// POUs/IO/Drives/SoE/Ax5000ParamSTRUCTs/P/AX5000_P_0270
{attribute 'pack_mode' := '1'}//Ensures 1-byte-alignmend
TYPE AX5000_P_0270 :
STRUCT
	Actual_lenght:UINT;
	Max_lenght:UINT;
	Feedback1:STRING(29);
//	{attribute 'hide'}
	Rsvd1:UINT;
	Serial_number_feedback1:ARRAY[0..1] OF UDINT;
	Feedback2:STRING(29);
//	{attribute 'hide'}
	Rsvd2:UINT;
	Serial_number_feedback2:ARRAY[0..1] OF UDINT;
	Modulo_value:UDINT;

(*Data read from file*)

(*data[0][0]*)
	Feedback_number1:UINT;
	Data_set1:UINT;
	Feedback_position1:UDINT;
	Modulo_position1:UDINT;
	Crc1:UDINT;
(*data[0][1]*)
	Feedback_number2:UINT;
	Data_se2t:UINT;
	Feedback_position2:UDINT;
	Modulo_position2:UDINT;
	Crc2:UDINT;
(*data[1][0]*)
	Feedback_number3:UINT;
	Data_set3:UINT;
	Feedback_position3:UDINT;
	Modulo_position3:UDINT;
	Crc3:UDINT;
(*data[1][1]*)
	Feedback_number4:UINT;
	Data_set4:UINT;
	Feedback_position4:UDINT;
	Modulo_position4:UDINT;
	Crc4:UDINT;


(*Current Data*)


(*data[0][0]*)
	Feedback_number5:UINT;
	Data_set5:UINT;
	Feedback_position5:UDINT;
	Modulo_position5:UDINT;
	Crc5:UDINT;
(*data[0][1]*)
	Feedback_number6:UINT;
	Data_se6t:UINT;
	Feedback_position6:UDINT;
	Modulo_position:UDINT;
	Crc6:UDINT;
(*data[1][0]*)
	Feedback_number7:UINT;
	Data_set7:UINT;
	Feedback_position7:UDINT;
	Modulo_position7:UDINT;
	Crc7:UDINT;
(*data[1][1]*)
	Feedback_number8:UINT;
	Data_set8:UINT;
	Feedback_position8:UDINT;
	Modulo_position8:UDINT;
	Crc8:UDINT;
END_STRUCT
END_TYPE

// POUs/IO/Drives/SoE/Ax5000ParamSTRUCTs/P/AX5000_P_0271
TYPE AX5000_P_0271 :
STRUCT
	Save_sosition_offset_pc:UINT;
END_STRUCT
END_TYPE

// POUs/IO/Drives/SoE/Ax5000ParamSTRUCTs/P/AX5000_P_0272
{attribute 'pack_mode' := '1'}//Ensures 1-byte-alignmend
TYPE AX5000_P_0272 :
STRUCT
	Actual_Length : UINT := 8;
	Max_Length : UINT := 8;
	(* FeedbackNumber &amp; MemorySelection *)
	Data : BYTE;
//	{attribute 'hide'}
	Rsvd1 : ARRAY [1..3] OF USINT;
	Position_Offset : UDINT;	
END_STRUCT
END_TYPE

// POUs/IO/Drives/SoE/Ax5000ParamSTRUCTs/P/AX5000_P_0273
TYPE AX5000_P_0273 EXTENDS ST_AX5000_P_0273:
STRUCT
(*
	Actual_lenght:UINT:= 112;
	Max_lenght:UINT := 112;
(*feedback 1*)
 {attribute 'GUID' := 'D1EB669D-3061-44CC-A2EE-FBF75E3AC2F6'}
 {attribute 'Namespace' := 'AX5000'}
Feedback1 : ST_AX5000_P_0273_Feedback;
(*
(*Encoder Memory*)
	Data_valid1:UINT;
//	{attribute 'hide'}
	rsvd1:UINT;
	Position_offset1:UDINT;
(*Drive Memory*)
	Data_valid2:UINT;
//	{attribute 'hide'}
	rsvd2:UINT;
	Feedback_type1:STRING(29);
//	{attribute 'hide'}
	rsvd3:UINT;
	Feedback_serial_number:ARRAY[0..1]OF UDINT;
	Position_offset2:UDINT;
*)
(*feedback 2*)
{attribute 'GUID' := 'D1EB669D-3061-44CC-A2EE-FBF75E3AC2F6'}
 {attribute 'Namespace' := 'AX5000'}
Feedback2 : ST_AX5000_P_0273_Feedback;
(*
(*Encoder Memory*)
	Data_valid3:UINT;
//	{attribute 'hide'}
	rsvd4:UINT;
	Position_offset3:UDINT;
(*Drive Memory*)
	Data_valid4:UINT;
//	{attribute 'hide'}
	rsvd5:UINT;
	Feedback_type2:STRING(29);
//	{attribute 'hide'}
	rsvd6:UINT;
	Feedback_serial_number2:ARRAY[0..1]OF UDINT;
	Position_offset4:UDINT;
*)	

//	{attribute 'hide'}
	Rsvd1 : UDINT;
*)
END_STRUCT
END_TYPE

// POUs/IO/Drives/SoE/Ax5000ParamSTRUCTs/P/AX5000_P_0274
{attribute 'pack_mode' := '1'}
TYPE AX5000_P_0274 :
STRUCT
	Actual_lenght:UINT;
	Max_lenght:UINT;
	Position_offset_feedback_1:UDINT;
	Position_offset_feedback_2:UDINT;
END_STRUCT
END_TYPE

// POUs/IO/Drives/SoE/Ax5000ParamSTRUCTs/P/AX5000_P_0275
TYPE AX5000_P_0275 EXTENDS ST_AX5000_P_0275: 
	STRUCT
(*		 {attribute 'GUID' := 'A39361D3-D4AC-4F67-8FEE-F366F3137B89'}
		 {attribute 'Namespace' := 'AX5000'}
		ActiveFeedbackAndMemory : E_AX5000_P_0275_ActiveFeedbackAndMemory;
		InitializationErrorBehavior : BIT;
		 {attribute 'hide'}
		_reserved1 : BIT;
		 {attribute 'hide'}
		_reserved2 : BIT;
		 {attribute 'hide'}
		_reserved3 : BIT;
		 {attribute 'hide'}
		_reserved4 : BIT;
		 {attribute 'hide'}
		_reserved5 : BIT;
		 {attribute 'hide'}
		_reserved6 : BIT;
		 {attribute 'hide'}
		_reserved7 : BIT;
*)
	END_STRUCT
END_TYPE

// POUs/IO/Drives/SoE/Ax5000ParamSTRUCTs/P/AX5000_P_0276
TYPE AX5000_P_0276 :
STRUCT
	Data_storage_feedback1_Data_storge_feedback2:UDINT;	(*Data_storage_feedback1 8Bit; Data_storage_feedback2 8 Bit*)
END_STRUCT
END_TYPE

// POUs/IO/Drives/SoE/Ax5000ParamSTRUCTs/P/AX5000_P_0277
TYPE AX5000_P_0277 :
STRUCT
	Schedule_modulo_init_data_saving:UINT;
END_STRUCT
END_TYPE

// POUs/IO/Drives/SoE/Ax5000ParamSTRUCTs/P/AX5000_P_0278
TYPE AX5000_P_0278 :
STRUCT
	Ignore_for_one_PreOp_SafeOp_transition:UINT;
END_STRUCT
END_TYPE

// POUs/IO/Drives/SoE/Ax5000ParamSTRUCTs/P/AX5000_P_0300
TYPE AX5000_P_0300 :
STRUCT
	Actual_lenght:UINT;
	Max_lenght:UINT;
	Error_number_history:ARRAY[0..99] OF UDINT;
END_STRUCT
END_TYPE

// POUs/IO/Drives/SoE/Ax5000ParamSTRUCTs/P/AX5000_P_0301
TYPE AX5000_P_0301 :
STRUCT
	Actual_lenght:UINT;
	Max_lenght:UINT;
	Error_times_history:ARRAY[0..99] OF UDINT;
END_STRUCT
END_TYPE

// POUs/IO/Drives/SoE/Ax5000ParamSTRUCTs/P/AX5000_P_0302
TYPE AX5000_P_0302 :
STRUCT
	Display_value_line_1:UINT;
END_STRUCT
END_TYPE

// POUs/IO/Drives/SoE/Ax5000ParamSTRUCTs/P/AX5000_P_0303
TYPE AX5000_P_0303 :
STRUCT
	Display_value_line_2:UINT;
END_STRUCT
END_TYPE

// POUs/IO/Drives/SoE/Ax5000ParamSTRUCTs/P/AX5000_P_0304
TYPE AX5000_P_0304 :
STRUCT
	Log_errors_Log_warnings_Log_information_rsvd:UINT;	(*Log_errors 1; BitLog_warnings 1; BitLog_information 1 Bit*)
END_STRUCT
END_TYPE

// POUs/IO/Drives/SoE/Ax5000ParamSTRUCTs/P/AX5000_P_0305
TYPE AX5000_P_0305 :
STRUCT
	I2C_Bus_Lcd_Ext_ADC_Encoder_parameter_channel_String_KeyPad_Procedure_command_calls_Powermanagement_Feedback_Dsp_Device_state_machine_rsvd:UDINT;
(*I2C_Bus 2 Bit; Lcd 2 Bit; Ext_ADC 2 Bit; Encoder 2 Bit; parameter_channel_String 2 Bit; KeyPad 2 Bit; Procedure_command_calls 2 Bit; Powermanagement 2 Bit; Feedback_Dsp 2 Bit; Device_state_machine 2 Bit; rsvd 12 Bit*)
END_STRUCT
END_TYPE

// POUs/IO/Drives/SoE/Ax5000ParamSTRUCTs/P/AX5000_P_0306
TYPE AX5000_P_0306 :
STRUCT
	Actual_main_loop_time:UINT;
END_STRUCT
END_TYPE

// POUs/IO/Drives/SoE/Ax5000ParamSTRUCTs/P/AX5000_P_0307
TYPE AX5000_P_0307 :
STRUCT
	Max_main_loop_time:UINT;
END_STRUCT
END_TYPE

// POUs/IO/Drives/SoE/Ax5000ParamSTRUCTs/P/AX5000_P_0308
TYPE AX5000_P_0308 :
STRUCT
	Actual_ctrl_loop_time:UINT;
END_STRUCT
END_TYPE

// POUs/IO/Drives/SoE/Ax5000ParamSTRUCTs/P/AX5000_P_0309
TYPE AX5000_P_0309 :
STRUCT
	Max_ctrl_loop_time:UINT;
END_STRUCT
END_TYPE

// POUs/IO/Drives/SoE/Ax5000ParamSTRUCTs/P/AX5000_P_0310
TYPE AX5000_P_0310 :
STRUCT
	Torque_off_Slow_down_according_Open_loop_ramp_Closed_loop_ramp_NC_handling_rsvd:UINT;
	(*Torque_off 1 Bit; Slow_down_according 1 Bit; Open_loop_ramp 1 Bit; Closed_loop_ramp 1 Bit; NC_handling  1 Bit;  rsvd  11 Bit; *)
END_STRUCT
END_TYPE

// POUs/IO/Drives/SoE/Ax5000ParamSTRUCTs/P/AX5000_P_0311
TYPE AX5000_P_0311 :
STRUCT
	PLL_ctrl_error:DINT;
END_STRUCT
END_TYPE

// POUs/IO/Drives/SoE/Ax5000ParamSTRUCTs/P/AX5000_P_0312
TYPE AX5000_P_0312 :
STRUCT
	PCB_temperature:UINT;
END_STRUCT
END_TYPE

// POUs/IO/Drives/SoE/Ax5000ParamSTRUCTs/P/AX5000_P_0313
TYPE AX5000_P_0313 :
STRUCT
	Actual_lenght:UINT;
	Max_lenght:UINT;
	String_output_mode:UINT;
	Backlight_mode:UINT;
	Keypad_mode:UINT;
//	{attribute 'hide'}
	Rsvd:UINT;
	Output_string:STRING(39);
END_STRUCT
END_TYPE

// POUs/IO/Drives/SoE/Ax5000ParamSTRUCTs/P/AX5000_P_0314
TYPE AX5000_P_0314 :
STRUCT
	Actual_lenght:UINT;
	Max_lenght:UINT;
	String_output_mode:UINT;
	Backlight_mode:UINT;
	Keypad_mode:UINT;
//	{attribute 'hide'}
	Rsvd:UINT;
	Output_string:STRING(39);
END_STRUCT
END_TYPE

// POUs/IO/Drives/SoE/Ax5000ParamSTRUCTs/P/AX5000_P_0315
TYPE AX5000_P_0315 :
STRUCT
	Configuration_Output_number_Set_output_error_Set_output_warning_rsvd:UINT;
	(*Configuration 3 Bit; Output_number 5 Bit; Set_output_error 1 Bit; Set_output_warning 1 Bit; rsvd 6 Bit; *)
END_STRUCT
END_TYPE

// POUs/IO/Drives/SoE/Ax5000ParamSTRUCTs/P/AX5000_P_0316
TYPE AX5000_P_0316 :
STRUCT
	Actual_lenght:UINT;
	Max_lenght:UINT;
	Mode:UINT;
	Level:UINT;		(*Decimal Point 1*)
END_STRUCT
END_TYPE

// POUs/IO/Drives/SoE/Ax5000ParamSTRUCTs/P/AX5000_P_0317
TYPE AX5000_P_0317 :
STRUCT
	Actual_amplifier_stilisation:UDINT;
END_STRUCT
END_TYPE

// POUs/IO/Drives/SoE/Ax5000ParamSTRUCTs/P/AX5000_P_0320
TYPE AX5000_P_0320 EXTENDS ST_AX5000_P_0320:
STRUCT
(*	Actual_lenght:UINT;
	Max_lenght:UINT;
	Firmware_version:UINT;
	Firmware_build:UINT;
	Bootloader_build:UINT;
	MainDsp_compiler_version:UDINT;
	FeedbackDsp_compiler_version:UDINT;
	Option_card_firmware_version:UINT;
	Option_card_firmware_build:UINT;
	Option_card_interface:UINT;
//	{attribute 'hide'}
	Rsvd:UDINT;
	Option_card_Dsp_compiler_version:UDINT;
	Intf_Build_Version:UINT;
//	{attribute 'hide'}
	Rsvd2:UINT;
//	{attribute 'hide'}
	Rsvd3:UINT;
*)
END_STRUCT
END_TYPE

// POUs/IO/Drives/SoE/Ax5000ParamSTRUCTs/P/AX5000_P_0321
{attribute 'pack_mode' := '1'}
TYPE AX5000_P_0321 :
STRUCT
	Actual_lenght:UINT;
	Max_lenght:UINT;
	Disc_size:UDINT;
	Usend_size:UDINT;
	Alignment:UDINT;
	Free_size:UDINT;
(*File 0*)
	Type0:UINT;
//	{attribute 'hide'}
	rsvd0:UINT;
	Version0:UINT;
	Build0:UINT;
	Time_H0:UDINT;
	Time_L0:UDINT;
	Id10:UINT;
	Id20:UINT;
	Size0:UDINT;
	Size_on_disk0:UDINT;
	alignment0:UDINT;
	Start_adresse0:UDINT;

(*File 1*)
	Type1:UINT;
//	{attribute 'hide'}
	Rsvd1:UINT;
	Version1:UINT;
	Build1:UINT;
	Time_H1:UDINT;
	Time_L1:UDINT;
	Id11:UINT;
	Id21:UINT;
	Size1:UDINT;
	Size_on_disk1:UDINT;
	alignment1:UDINT;
	Start_adresse1:UDINT;

(*File 2*)
	Type2:UINT;
//	{attribute 'hide'}
	Rsvd2:UINT;
	Version2:UINT;
	Build2:UINT;
	Time_H2:UDINT;
	Time_L2:UDINT;
	Id12:UINT;
	Id22:UINT;
	Size2:UDINT;
	Size_on_disk2:UDINT;
	alignment2:UDINT;
	Start_adresse2:UDINT;

(*File 3*)
	Type3:UINT;
//	{attribute 'hide'}
	Rsvd3:UINT;
	Version3:UINT;
	Build3:UINT;
	Time_H3:UDINT;
	Time_L3:UDINT;
	Id13:UINT;
	Id23:UINT;
	Size3:UDINT;
	Size_on_disk3:UDINT;
	alignment3:UDINT;
	Start_adresse3:UDINT;

(*File 4*)
	Type4:UINT;
//	{attribute 'hide'}
	Rsvd4:UINT;
	Version4:UINT;
	Build4:UINT;
	Time_H4:UDINT;
	Time_L4:UDINT;
	Id14:UINT;
	Id24:UINT;
	Size4:UDINT;
	Size_on_disk4:UDINT;
	alignment4:UDINT;
	Start_adresse4:UDINT;

(*File 5*)
	Type5:UINT;
//	{attribute 'hide'}
	Rsvd5:UINT;
	Version5:UINT;
	Build5:UINT;
	Time_H5:UDINT;
	Time_L5:UDINT;
	Id15:UINT;
	Id25:UINT;
	Size5:UDINT;
	Size_on_disk5:UDINT;
	alignment5:UDINT;
	Start_adresse5:UDINT;

(*File 6*)
	Type6:UINT;
//	{attribute 'hide'}
	Rsvd6:UINT;
	Version6:UINT;
	Build6:UINT;
	Time_H6:UDINT;
	Time_L6:UDINT;
	Id16:UINT;
	Id26:UINT;
	Size6:UDINT;
	Size_on_disk6:UDINT;
	alignment6:UDINT;
	Start_adresse6:UDINT;

(*File 7*)
	Type7:UINT;
//	{attribute 'hide'}
	Rsvd7:UINT;
	Version7:UINT;
	Build7:UINT;
	Time_H7:UDINT;
	Time_L7:UDINT;
	Id17:UINT;
	Id27:UINT;
	Size7:UDINT;
	Size_on_disk7:UDINT;
	Alignment7:UDINT;
	Start_adresse7:UDINT;

(*File 8*)
	Type8:UINT;
//	{attribute 'hide'}
	Rsvd8:UINT;
	Version8:UINT;
	Build8:UINT;
	Time_H8:UDINT;
	Time_L8:UDINT;
	Id18:UINT;
	Id28:UINT;
	Size8:UDINT;
	Size_on_disk8:UDINT;
	Alignment8:UDINT;
	Start_adresse8:UDINT;

(*File 9*)
	Type9:UINT;
	Rsvd9:UINT;
	Version9:UINT;
	Build9:UINT;
	Time_H9:UDINT;
	Time_L9:UDINT;
	Id19:UINT;
	Id29:UINT;
	Size9:UDINT;
	Size_on_disk9:UDINT;
	alignment9:UDINT;
	Start_adresse9:UDINT;
END_STRUCT
END_TYPE

// POUs/IO/Drives/SoE/Ax5000ParamSTRUCTs/P/AX5000_P_0322
//	{attribute 'hide'}
TYPE AX5000_P_0322 :
STRUCT
	Actual_lenght:UINT;
	Max_lenght:UINT;


	PCB_ID_version:UINT;
	Hwld1:UINT;
	Hwld2:UINT;
	Hwld3:UINT;
	Manufacturing_Data:UINT;
	Serial_number_low:UINT;
	Serial_number_high:UINT;
	Checksum:UINT;


	PCB_ID_version1:UINT;
	Hwld4:UINT;
	Hwld5:UINT;
	Hwld6:UINT;
	Manufacturing_Data1:UINT;
	Serial_number_low1:UINT;
	Serial_number_high1:UINT;
	Checksum1:UINT;


	PCB_ID_version2:UINT;
	Hwld7:UINT;
	Hwld8:UINT;
	Hwld9:UINT;
	Manufacturing_Data2:UINT;
	Serial_number_low2:UINT;
	Serial_number_high2:UINT;
	Checksum2:UINT;


	PCB_ID_version3:UINT;
	Hwld10:UINT;
	Hwld11:UINT;
	Hwld12:UINT;
	Manufacturing_Data3:UINT;
	Serial_number_low3:UINT;
	Serial_number_high3:UINT;
	Checksum3:UINT;


	PCB_ID_version4:UINT;
	Hwld13:UINT;
	Hwld14:UINT;
	Hwld15:UINT;
	Manufacturing_Data4:UINT;
	Serial_number_low4:UINT;
	Serial_number_high4:UINT;
	Checksum4:UINT;


	PCB_ID_version5:UINT;
	Hwld16:UINT;
	Hwld17:UINT;
	Hwld18:UINT;
	Manufacturing_Data5:UINT;
	Serial_number_low5:UINT;
	Serial_number_high5:UINT;
	Checksum5:UINT;


	Control_Pcb_Id_valid:UINT;
	Power_Pcb_Id_valid:UINT;
	Driver_Pcb_Id_valid:UINT;
	Front_Pcb_Id_valid:UINT;
	OptionSlot_Pcb_Id_valid:UINT;
	SafetySlot_Id_valid:UINT;
	Dsp_Revidion:UINT;
	Dsp_Id_Xint_Revision:UINT;
	Feedback_Dsp_Id:UINT;
	Feedback_Dsp_Revision:UINT;
	Esc_Revision:UINT;
	Esc_build:UINT;
	Esc_type:UINT;
	FPGA_device_Type:UINT;
	FPGA_device_Subtype:UINT;
	FPGA_version_number:UINT;
	FPGA_build_number:UINT;
	Option_slot_FPGA:UINT;
END_STRUCT
END_TYPE

// POUs/IO/Drives/SoE/Ax5000ParamSTRUCTs/P/AX5000_P_0323
TYPE AX5000_P_0323 :
STRUCT
	Actual_lenght:UINT;
	Max_lenght:UINT;

(*control*)
	Total:UDINT;
	Available:UDINT;
	Total1:UDINT;
	Available1:UDINT;
	Total2:UDINT;
	Available2:UDINT;
	Total3:UDINT;
	Available3:UDINT;

(*front*)
	Total4:UDINT;
	Available4:UDINT;
	Total5:UDINT;
	Available5:UDINT;
	Total6:UDINT;
	Available6:UDINT;
	Total7:UDINT;
	Available7:UDINT;


(*option*)
	Toal8:UDINT;
	Available8:UDINT;
	Total9:UDINT;
	Available9:UDINT;
	Total10:UDINT;
	Available10:UDINT;
	Total11:UDINT;
	Available11:UDINT;
END_STRUCT
END_TYPE

// POUs/IO/Drives/SoE/Ax5000ParamSTRUCTs/P/AX5000_P_0324
TYPE AX5000_P_0324 :
STRUCT
	Actual_lenght:UINT;
	Max_lenght:UINT;
	ProductCode_RevisionNo:STRING;
END_STRUCT
END_TYPE

// POUs/IO/Drives/SoE/Ax5000ParamSTRUCTs/P/AX5000_P_0325
TYPE AX5000_P_0325 :
STRUCT
	Actual_lenght:UINT;
	Max_lenght:UINT;
	Compile_time_and_date:STRING;
END_STRUCT
END_TYPE

// POUs/IO/Drives/SoE/Ax5000ParamSTRUCTs/P/AX5000_P_0326
TYPE AX5000_P_0326 :
STRUCT
	Actual_lenght:UINT;
	Max_lenght:UINT;
	Release_note:STRING;
END_STRUCT
END_TYPE

// POUs/IO/Drives/SoE/Ax5000ParamSTRUCTs/P/AX5000_P_0350
TYPE AX5000_P_0350 EXTENDS ST_AX5000_P_0350: 
STRUCT
//	Error_reaction_Controlword:UINT;
END_STRUCT
END_TYPE

// POUs/IO/Drives/SoE/Ax5000ParamSTRUCTs/P/AX5000_P_0351
TYPE AX5000_P_0351 :
STRUCT
	Error_reaktion_delay_time:UINT;
END_STRUCT
END_TYPE

// POUs/IO/Drives/SoE/Ax5000ParamSTRUCTs/P/AX5000_P_0352
TYPE AX5000_P_0352 :
STRUCT
	Drive_halt_jerk_bipolar:UDINT;
END_STRUCT
END_TYPE

// POUs/IO/Drives/SoE/Ax5000ParamSTRUCTs/P/AX5000_P_0353
TYPE AX5000_P_0353 :
STRUCT
	Emergency_stop_jerk:UDINT;
END_STRUCT
END_TYPE

// POUs/IO/Drives/SoE/Ax5000ParamSTRUCTs/P/AX5000_P_0354
TYPE AX5000_P_0354 :
STRUCT
	Standstill_window_monitoring_time:UINT;
END_STRUCT
END_TYPE

// POUs/IO/Drives/SoE/Ax5000ParamSTRUCTs/P/AX5000_P_0356
//	{attribute 'hide'}
TYPE AX5000_P_0356 :
STRUCT
	Actual_lenght:UINT;
	Max_lenght:UINT;
//	{attribute 'hide'}
	Rsvd:UDINT;
	Available_for:UINT;
	Command_mode:UINT;
	Current_level:UINT;
	Current_slope:UINT;
	Wait_time_before_braking:UINT;
	First_phase_activation_time_with_f_f1:UINT;
	Rotary_field_frequency_f1:UINT;
	Rotor_slowdown_mode:UINT;
	Second_phase_activation_time_with_f_0Hz:UINT;
	Wait_ime_after_braking:UINT;
//	{attribute 'hide'}
	Rsvd1:UINT;
//	{attribute 'hide'}
	Rsvd2:UINT;
	Synchronus_motor:ARRAY[0..11] OF UINT;
END_STRUCT
END_TYPE

// POUs/IO/Drives/SoE/Ax5000ParamSTRUCTs/P/AX5000_P_0360
TYPE AX5000_P_0360 :
STRUCT
	Parameter_set_prearrangement:UINT;
END_STRUCT
END_TYPE

// POUs/IO/Drives/SoE/Ax5000ParamSTRUCTs/P/AX5000_P_0361
TYPE AX5000_P_0361 :
STRUCT
	Actual_lenght:UINT;
	Max_lenght:UINT;
	Parameter_set_configuration:ARRAY[0..34] OF UINT;
END_STRUCT
END_TYPE

// POUs/IO/Drives/SoE/Ax5000ParamSTRUCTs/P/AX5000_P_0400
TYPE AX5000_P_0400 EXTENDS ST_AX5000_P_0400:
STRUCT
//	Hardware_enable_configuration:UINT;
END_STRUCT
END_TYPE

// POUs/IO/Drives/SoE/Ax5000ParamSTRUCTs/P/AX5000_P_0401
TYPE AX5000_P_0401 :
STRUCT
	Positiv_limit_switch: ST_AX5000_P_0401_LimitSwitch;
	Negativ_limit_switch: ST_AX5000_P_0401_LimitSwitch;
END_STRUCT
END_TYPE

// POUs/IO/Drives/SoE/Ax5000ParamSTRUCTs/P/AX5000_P_0402
TYPE AX5000_P_0402 :
STRUCT
	Redy_to_operate_configuration:UINT;
END_STRUCT
END_TYPE

// POUs/IO/Drives/SoE/Ax5000ParamSTRUCTs/P/AX5000_P_0451
TYPE AX5000_P_0451 :
STRUCT
	Current_controller_settings:UINT;
END_STRUCT
END_TYPE

// POUs/IO/Drives/SoE/Ax5000ParamSTRUCTs/P/AX5000_P_0452
TYPE AX5000_P_0452 :
STRUCT
	Current_controller_control_word:UINT;
END_STRUCT
END_TYPE

// POUs/IO/Drives/SoE/Ax5000ParamSTRUCTs/P/AX5000_P_0453
TYPE AX5000_P_0453 :
STRUCT
	Current_controller_status_word:UINT;
END_STRUCT
END_TYPE

// POUs/IO/Drives/SoE/Ax5000ParamSTRUCTs/P/AX5000_P_0454
TYPE AX5000_P_0454 :
STRUCT
	Effective_torque_command_value:UINT;
END_STRUCT
END_TYPE

// POUs/IO/Drives/SoE/Ax5000ParamSTRUCTs/P/AX5000_P_0455
{attribute 'pack_mode' := '1'}
TYPE AX5000_P_0455 :
STRUCT
	Actual_lenght:UINT;
	Max_lenght:UINT;
	Mode:UINT;
	Rsvd:UINT;
	Min_voltage:UINT;
	Max_voltage:UINT;
	Max_current_for_fielweakening:UDINT;
	Max_velocity_for_fielweakening:UDINT;
END_STRUCT
END_TYPE

// POUs/IO/Drives/SoE/Ax5000ParamSTRUCTs/P/AX5000_P_0456
TYPE AX5000_P_0456 :
STRUCT
	Actual_motor_voltage_phase_U:UINT;
END_STRUCT
END_TYPE

// POUs/IO/Drives/SoE/Ax5000ParamSTRUCTs/P/AX5000_P_0457
TYPE AX5000_P_0457 :
STRUCT
	Actual_motor_voltage_phase_V:UINT;
END_STRUCT
END_TYPE

// POUs/IO/Drives/SoE/Ax5000ParamSTRUCTs/P/AX5000_P_0458
TYPE AX5000_P_0458 :
STRUCT
	Actual_motor_voltage_phase_W:UINT;
END_STRUCT
END_TYPE

// POUs/IO/Drives/SoE/Ax5000ParamSTRUCTs/P/AX5000_P_0459
TYPE AX5000_P_0459 :
STRUCT
	Actual_torquw_generating_current:UINT;
END_STRUCT
END_TYPE

// POUs/IO/Drives/SoE/Ax5000ParamSTRUCTs/P/AX5000_P_0460
TYPE AX5000_P_0460 :
STRUCT
	Actual_flux_generating_current:UINT;
END_STRUCT
END_TYPE

// POUs/IO/Drives/SoE/Ax5000ParamSTRUCTs/P/AX5000_P_0461
TYPE AX5000_P_0461 :
STRUCT
	Actual_absolute_current:UINT;
END_STRUCT
END_TYPE

// POUs/IO/Drives/SoE/Ax5000ParamSTRUCTs/P/AX5000_P_0462
TYPE AX5000_P_0462 :
STRUCT
	Actual_peak_current_limit:UINT;
END_STRUCT
END_TYPE

// POUs/IO/Drives/SoE/Ax5000ParamSTRUCTs/P/AX5000_P_0463
TYPE AX5000_P_0463 :
STRUCT
	Actual_current_limit:UINT;
END_STRUCT
END_TYPE

// POUs/IO/Drives/SoE/Ax5000ParamSTRUCTs/P/AX5000_P_0464
{attribute 'pack_mode' := '1'}
TYPE AX5000_P_0464 :
STRUCT
	Actual_lenght:UINT;
	Max_lenght:UINT;
	Mode:UINT;
	Adaptive_gain:UINT;
	Min_bandswitch:UINT;
	Max_bandswitch:UINT;
	Correction_factor_Iq_to_Acc:UINT;
	Damping:UINT;
	Starting_current_command:UINT;
	Rsvd:UINT;
	Threshold_speed1:UDINT;
	Threshold_speed2:UDINT;
//	{attribute 'hide'}
	Rsvd2:UDINT;
END_STRUCT
END_TYPE

// POUs/IO/Drives/SoE/Ax5000ParamSTRUCTs/P/AX5000_P_0502
TYPE AX5000_P_0502 :
STRUCT
	Velocity_controller_control_word:UINT;
END_STRUCT
END_TYPE

// POUs/IO/Drives/SoE/Ax5000ParamSTRUCTs/P/AX5000_P_0503
TYPE AX5000_P_0503 :
STRUCT
	Velocity_controller_status_word:UINT;
END_STRUCT
END_TYPE

// POUs/IO/Drives/SoE/Ax5000ParamSTRUCTs/P/AX5000_P_0504
TYPE AX5000_P_0504 :
STRUCT
	Effective_velocity_command_value:UDINT;
END_STRUCT
END_TYPE

// POUs/IO/Drives/SoE/Ax5000ParamSTRUCTs/P/AX5000_P_0505
TYPE AX5000_P_0505 :
STRUCT
	Velocity_controller_output:UINT;
END_STRUCT
END_TYPE

// POUs/IO/Drives/SoE/Ax5000ParamSTRUCTs/P/AX5000_P_0511
TYPE AX5000_P_0511 :
STRUCT
	Celocity_filter_low_pass_time_constant:UINT;
END_STRUCT
END_TYPE

// POUs/IO/Drives/SoE/Ax5000ParamSTRUCTs/P/AX5000_P_0512
TYPE AX5000_P_0512 :
STRUCT
	Velocity_filter_low_pass_damping:UDINT;
END_STRUCT
END_TYPE

// POUs/IO/Drives/SoE/Ax5000ParamSTRUCTs/P/AX5000_P_0513
{attribute 'pack_mode' := '1'}
TYPE AX5000_P_0513 :
STRUCT
	Actual_lenght:UINT;
	Max_lenght:UINT;
	ST_CONV_Version:UINT;
	Rsvd1:UINT;
	Filter_type:UINT;
//	{attribute 'hide'}
	nRsvd2:UINT;
	Low_pass_frequency:UDINT;
	Low_pass_damping:UDINT;
	High_pass_frequency:UDINT;
	High_pass_damping:UDINT;
//	{attribute 'hide'}
	Rsvd3:UDINT;
//	{attribute 'hide'}
	Rsvd4:UDINT;
	QMath_factor:UINT;
//	{attribute 'hide'}
	nRsvd5:UINT;
	b0:UDINT;
	b1:UDINT;
	b2:UDINT;
	a1:UDINT;
	a2:UDINT;
//	{attribute 'hide'}
	Rsvd6:UDINT;
	Rsvd7:UDINT;
END_STRUCT
END_TYPE

// POUs/IO/Drives/SoE/Ax5000ParamSTRUCTs/P/AX5000_P_0514
{attribute 'pack_mode' := '1'}
TYPE AX5000_P_0514 :
STRUCT
	Actual_lenght:UINT;
	Max_lenght:UINT;
	Mode:UINT;
//	{attribute 'hide'}
	Rsvd1:UINT;
	Bandswitch:UINT;
	Correction_factor_Iq_to_acc:UINT;
	Damping:UINT;
//	{attribute 'hide'}
	Rsvd2:UINT;
END_STRUCT
END_TYPE

// POUs/IO/Drives/SoE/Ax5000ParamSTRUCTs/P/AX5000_P_0515
{attribute 'pack_mode' := '1'}
TYPE AX5000_P_0515 :
STRUCT
	Actual_lenght:UINT;
	Max_lenght:UINT;
	ST_CONV_Version:UINT;
//	{attribute 'hide'}
	Rsvd1:UINT;
	Filter_type:UINT;
//	{attribute 'hide'}
	Rsvd2:UINT;
	Low_pass_frequency:UDINT;
	Low_pass_damping:UDINT;
	High_pass_frequency:UDINT;
	High_pass_damping:UDINT;
//	{attribute 'hide'}
	Rsvd3:UDINT;
//	{attribute 'hide'}
	Rsvd4:UDINT;
	QMath_factor:UINT;
//	{attribute 'hide'}
	Rsvd5:UINT;
	b0:UDINT;
	b1:UDINT;
	b2:UDINT;
	a1:UDINT;
	a2:UDINT;
//	{attribute 'hide'}
	Rsvd6:UDINT;
//	{attribute 'hide'}
	Rsvd7:UDINT;
END_STRUCT
END_TYPE

// POUs/IO/Drives/SoE/Ax5000ParamSTRUCTs/P/AX5000_P_0516
{attribute 'pack_mode' := '1'}
TYPE AX5000_P_0516 :
STRUCT
	Actual_lenght:UINT;
	Max_lenght:UINT;
	ST_CONV_Version:UINT;
	Rsvd1:UINT;
	Filter_type:UINT;
//	{attribute 'hide'}
	Rsvd2:UINT;
	Low_pass_frequency:UDINT;
	Low_pass_damping:UDINT;
	High_pass_frequency:UDINT;
	High_pass_damping:UDINT;
//	{attribute 'hide'}
	Rsvd3:UDINT;
//	{attribute 'hide'}
	Rsvd4:UDINT;
	QMath_factor:UINT;
//	{attribute 'hide'}
	Rsvd5:UINT;
	b0:UDINT;
	b1:UDINT;
	b2:UDINT;
	a1:UDINT;
	a2:UDINT;
//	{attribute 'hide'}
	Rsvd6:UDINT;
	Rsvd7:UDINT;
END_STRUCT
END_TYPE

// POUs/IO/Drives/SoE/Ax5000ParamSTRUCTs/P/AX5000_P_0517
{attribute 'pack_mode' := '1'}
TYPE AX5000_P_0517 :
STRUCT
	Actual_lenght:UINT;
	Max_lenght:UINT;
	ST_CONV_Version:UINT;
//	{attribute 'hide'}
	Rsvd1:UINT;
	Filter_type:UINT;
//	{attribute 'hide'}
	Rsvd2:UINT;
	Low_pass_frequency:UDINT;
	Low_pass_damping:UDINT;
	High_pass_frequency:UDINT;
	High_pass_damping:UDINT;
//	{attribute 'hide'}
	Rsvd3:UDINT;
//	{attribute 'hide'}
	nRsvd4:UDINT;
	QMath_factor:UINT;
	Rsvd5:UINT;
	b0:UDINT;
	b1:UDINT;
	b2:UDINT;
	a1:UDINT;
	a2:UDINT;
//	{attribute 'hide'}
	Rsvd6:UDINT;
//	{attribute 'hide'}
	Rsvd7:UDINT;
END_STRUCT
END_TYPE

// POUs/IO/Drives/SoE/Ax5000ParamSTRUCTs/P/AX5000_P_0518
{attribute 'pack_mode' := '1'}
TYPE AX5000_P_0518 :
STRUCT
	Actual_lenght:UINT;
	Max_lenght:UINT;
	Mode:UINT;
//	{attribute 'hide'}
	Rsvd:UINT;
	Velocity_window:UDINT;
	TIME_:UINT;
//	{attribute 'hide'}
	Rsvd1:UINT;
//	{attribute 'hide'}
	Rsvd2:UINT;
//	{attribute 'hide'}
	Rsvd3:UINT;
END_STRUCT
END_TYPE

// POUs/IO/Drives/SoE/Ax5000ParamSTRUCTs/P/AX5000_P_0552
TYPE AX5000_P_0552 :
STRUCT
	Position_controller_word:UINT;
END_STRUCT
END_TYPE

// POUs/IO/Drives/SoE/Ax5000ParamSTRUCTs/P/AX5000_P_0553
TYPE AX5000_P_0553 :
STRUCT
	Position_controller_status_word:UINT;
END_STRUCT
END_TYPE

// POUs/IO/Drives/SoE/Ax5000ParamSTRUCTs/P/AX5000_P_0554
TYPE AX5000_P_0554 :
STRUCT
	Effective_position_command_value:DINT;
END_STRUCT
END_TYPE

// POUs/IO/Drives/SoE/Ax5000ParamSTRUCTs/P/AX5000_P_0555
TYPE AX5000_P_0555 :
STRUCT
	Position_command_value_monitoring_window:UINT;
END_STRUCT
END_TYPE

// POUs/IO/Drives/SoE/Ax5000ParamSTRUCTs/P/AX5000_P_0556
TYPE AX5000_P_0556 :
STRUCT
	Position_interpolator_type:UINT;
END_STRUCT
END_TYPE

// POUs/IO/Drives/SoE/Ax5000ParamSTRUCTs/P/AX5000_P_0557
TYPE AX5000_P_0557 :
STRUCT
	Acceleration_feedforward_filter_timeconstant:UINT;
END_STRUCT
END_TYPE

// POUs/IO/Drives/SoE/Ax5000ParamSTRUCTs/P/AX5000_P_0558
TYPE AX5000_P_0558 :
STRUCT
	Position_controller_output:DINT;
END_STRUCT
END_TYPE

// POUs/IO/Drives/SoE/Ax5000ParamSTRUCTs/P/AX5000_P_0601
TYPE AX5000_P_0601 :
STRUCT
	Predictive_velocity_command_value:DINT;
END_STRUCT
END_TYPE

// POUs/IO/Drives/SoE/Ax5000ParamSTRUCTs/P/AX5000_P_0602
TYPE AX5000_P_0602 :
STRUCT
	Predictive_torque_command_value:INT;
END_STRUCT
END_TYPE

// POUs/IO/Drives/SoE/Ax5000ParamSTRUCTs/P/AX5000_P_0610
{attribute 'pack_mode' := '1'}
TYPE AX5000_P_0610 :
STRUCT
	Actual_lenght:UINT;
	Max_lenght:UINT;
	Velocity_limit:DINT;
	Velocity_condition:UINT;
//	{attribute 'hide'}
	Rsvd:UINT;
	Torque_force_limit:UINT;
//	{attribute 'hide'}
	Rsvd1:UINT;
	Torque_force_condition:UINT;
//	{attribute 'hide'}
	Rsvd2:UINT;
//	{attribute 'hide'}
	Rsvd3:UDINT;
//	{attribute 'hide'}
	Rsvd4:UDINT;
END_STRUCT
END_TYPE

// POUs/IO/Drives/SoE/Ax5000ParamSTRUCTs/P/AX5000_P_0611
TYPE AX5000_P_0611 :
STRUCT
	Configurable_status_word:UINT;
END_STRUCT
END_TYPE

// POUs/IO/Drives/SoE/Ax5000ParamSTRUCTs/P/AX5000_P_0800
TYPE AX5000_P_0800 :
STRUCT
	Digital_output_control_word:UINT;
END_STRUCT
END_TYPE

// POUs/IO/Drives/SoE/Ax5000ParamSTRUCTs/P/AX5000_P_0801
TYPE AX5000_P_0801 :
STRUCT
	Digital_inputs_state:UINT;
END_STRUCT
END_TYPE

// POUs/IO/Drives/SoE/Ax5000ParamSTRUCTs/P/AX5000_P_0802
TYPE AX5000_P_0802 :
STRUCT
	Digital_output:UINT;
END_STRUCT
END_TYPE

// POUs/IO/Drives/SoE/Ax5000ParamSTRUCTs/P/AX5000_P_0804
TYPE AX5000_P_0804 :
STRUCT
	Digital_feedback_inputs_option_unit:UINT;
END_STRUCT
END_TYPE

// POUs/IO/Drives/SoE/Ax5000ParamSTRUCTs/P/AX5000_P_0805
TYPE AX5000_P_0805 :
STRUCT
	Force_digital_inputs:UDINT;
END_STRUCT
END_TYPE

// POUs/IO/Drives/SoE/Ax5000ParamSTRUCTs/P/AX5000_P_0806
TYPE AX5000_P_0806 :
STRUCT
	Amplifier_output_voltage_slope:INT;
END_STRUCT
END_TYPE

// POUs/IO/Drives/SoE/Ax5000ParamSTRUCTs/P/AX5000_P_0810
TYPE AX5000_P_0810 :
STRUCT
	Actual_lenght:UINT;
	Max_lenght:UINT;
	Funktion_number:UDINT;
	Code_word:UDINT;
	Parameter1:UDINT;
	Parameter2:UDINT;
	Parameter3:UDINT;
	Parameter4:UDINT;
	Parameter5:UDINT;

END_STRUCT
END_TYPE

// POUs/IO/Drives/SoE/Ax5000ParamSTRUCTs/P/AX5000_P_0811
TYPE AX5000_P_0811 :
STRUCT
	Customer_specific_functionality_status:UDINT;
END_STRUCT
END_TYPE

// POUs/IO/Drives/SoE/Ax5000ParamSTRUCTs/P/AX5000_P_0850
TYPE AX5000_P_0850 :
STRUCT
	Actual_lenght:UINT;
	Max_lenght:UINT;
	Amplifier_identification:STRING(63);
END_STRUCT
END_TYPE

// POUs/IO/Drives/SoE/Ax5000ParamSTRUCTs/P/AX5000_P_0851
TYPE AX5000_P_0851 :
STRUCT
	Save_amplifier_identification:UINT;
END_STRUCT
END_TYPE

// POUs/IO/Drives/SoE/Ax5000ParamSTRUCTs/P/AX5000_P_0900
TYPE AX5000_P_0900 :
STRUCT
	Actual_lenght:UINT;
	Max_lenght:UINT;
(*Control Pcb*)
	Safety_test_status:UINT;
//	{attribute 'hide'}
	Rsvd1:UINT;
	Channel0_offset:INT;
	Channel0_gain:UINT;
	Channel1_offset:INT;
	Channel1_gain:UINT;
	Channel2_offset:INT;
	Channel2_gain:UINT;
	Channel3_offset:INT;
	Channel3_gain:UINT;
	Channel4_offset:INT;
	Channel4_gain:UINT;
	Channel5_offset:INT;
	Channel5_gain:UINT;
	Channel6_offset:INT;
	Channel6_gain:UINT;
	Channel7_offset:INT;
	Channel7_gain:UINT;
	Channel8_offset:INT;
	Channel8_gain:UINT;
	Channel9_offset:INT;
	Channel9_gain:UINT;
//	{attribute 'hide'}
	Rsvd2:ARRAY[0..6] OF UINT;
	Checksum:UINT;

(*Power Pcb*)
	(*Ch A*)
	ChA_Calibration_type:UINT;
	ChA_V_Offset:INT;
	ChA_W_Offset:INT;
	ChA_V_resistor_value1:UINT;
	ChA_W_resistor_value1:UINT;
	ChA_V_resistor_value2:UINT;
	ChA_W_resistor_value2:UINT;
	ChA_V_resistor_value3:UINT;
	ChA_W_resistor_value3:UINT;
	ChA_V_resistor_value4:UINT;
	ChA_W_resistor_value4:UINT;
	ChA_V_current_value1:UINT;
	ChA_W_current_value1:UINT;
	ChA_V_current_value2:UINT;
	ChA_W_current_value2:UINT;
	ChA_V_current_value3:UINT;
	ChA_W_current_value3:UINT;
	ChA_V_current_value4:UINT;
	ChA_W_current_value4:UINT;
	(*Ch B*)
	ChB_Calibration_type:UINT;
	ChB_V_Offset:INT;
	ChB_W_Offset:INT;
	ChB_V_resistor_value1:UINT;
	ChB_W_resistor_value1:UINT;
	ChB_V_resistor_value2:UINT;
	ChB_W_resistor_value2:UINT;
	ChB_V_resistor_value3:UINT;
	ChB_W_resistor_value3:UINT;
	ChB_V_resistor_value4:UINT;
	ChB_W_resistor_value4:UINT;
	ChB_V_current_value1:UINT;
	ChB_W_current_value1:UINT;
	ChB_V_current_value2:UINT;
	ChB_W_current_value2:UINT;
	ChB_V_current_value3:UINT;
	ChB_W_current_value3:UINT;
	ChB_V_current_value4:UINT;
	ChB_W_current_value4:UINT;
//	{attribute 'hide'}
	Rsvd3:UINT;
	Checksum2:UINT;

(*Driver Pcb*)
	Safety_test_status2:UINT;
	Calibration_type2:UINT;
//	{attribute 'hide'}
	Rsvd4:UINT;
	Udclink_offset:UINT;
	Udclink_gain:UINT;
	Udclink_offset1:UINT;
	Udclink_gain1:UINT;
	Udclink_offset2:UINT;
	Udclink_gain2:UINT;
	Udclink_offset3:UINT;
	Udclink_gain3:UINT;
//	{attribute 'hide'}
	Rsvd5:ARRAY[0..17] OF UINT;
	Checksum3:UINT;

(*Front Pcb*)
	Vendor:UDINT;
	Product_code:UDINT;
	Revision_No:UDINT;
	Serial_No:UDINT;
	Year:USINT;
	Week:USINT;
	Fan_profiltype_internalbrakeresistor_rsvd:UINT;		(*jeweils 4 Bit*)
	Hardware_device_id_2:UINT;
	Hardware_device_id_3:UINT;
	Hardware_device_id_4:UINT;
//	{attribute 'hide'}
	Rsvd6:ARRAY[0..2] OF UINT;
	Customized_id:UINT;
	ModificationId:UINT;
//	{attribute 'hide'}
	Rsvd7:ARRAY[0..3] OF UINT;
	Free_switch_code1:UINT;
	Free_switch_code2:UINT;
//	{attribute 'hide'}
	Rsvd8:ARRAY[0..3] OF UINT;
	ST_CONV_Version:UINT;
//	{attribute 'hide'}
	Rsvd9:UINT;
	(*ChA*)
	ChA_Sin_offset:DINT;
	ChA_Cos_offset:DINT;
	ChA_Sin_gain:UDINT;
	ChA_Cos_gain:UDINT;
	ChA_Excitation_voltage_Gain:UINT;
	ChA_rsvd10:ARRAY[0..2] OF UINT;
	(*ChB*)
	ChB_Sin_offset:DINT;
	ChB_Cos_offset:DINT;
	ChB_Sin_gain:UDINT;
	ChB_Cos_gain:UDINT;
	ChB_Excitation_voltage_Gain:UINT;
	ChB_rsvd11:ARRAY[0..2] OF UINT;
//{attribute 'hide'}
	Rsvd12:ARRAY[0..24] OF UINT;
	Checksum4:UINT;

(*Option Pcb*)
	Vendor2:UDINT;
	Product_code2:UDINT;
	Revision_No2:UDINT;
	Serial_No2:UDINT;
	Year2:USINT;
	Week2:USINT;
	Fan_profiltype_internalbrakeresistor_rsvd2:UINT;		(*jeweils 4 Bit*)
	Hardware_device_id_22:UINT;
	Hardware_device_id_32:UINT;
	Hardware_device_id_42:UINT;
//	{attribute 'hide'}
	Rsvd13:ARRAY[0..2] OF UINT;
	Customized_id2:UINT;
	ModificationId2:UINT;
//	{attribute 'hide'}
	Rsvd14:ARRAY[0..3] OF UINT;
	Free_switch_code12:UINT;
	Free_switch_code22:UINT;
//	{attribute 'hide'}
	Rsvd15:ARRAY[0..3] OF UINT;
	Version2:UINT;
//	{attribute 'hide'}
	Rsvd16:UINT;
	(*ChA*)
	ChA_Sin_offset2:DINT;
	ChA_Cos_offset2:DINT;
	ChA_Sin_gain2:UDINT;
	ChA_Cos_gain2:UDINT;
	ChA_Excitation_voltage_Gai2n:UINT;
	ChA_rsvd17:ARRAY[0..2] OF UINT;
	(*ChB*)
	ChB_Sin_offset2:DINT;
	ChB_Cos_offse2t:DINT;
	ChB_Sin_gain2:UDINT;
	ChB_Cos_gain2:UDINT;
	ChB_Excitation_voltage_Gai2n:UINT;
	ChB_rsvd18:ARRAY[0..2] OF UINT;
//{attribute 'hide'}
	Rsvd19:ARRAY[0..24] OF UINT;
	Checksum5:UINT;

(*Safety Pcb*)
//{attribute 'hide'}
	Rsvd20:ARRAY[0..8] OF UINT;
	Checksum6:UINT;

	Control_Pcb_data_valid:UINT;
	Power_Pcb_data_valid:UINT;
	Driver_Pcb_data_valid:UINT;
	Front_Pcb_data_valid:UINT;
	Option_Pcb_data_valid:UINT;
	Safety_Pcb_data_valid:UINT;

END_STRUCT
END_TYPE

// POUs/IO/Drives/SoE/Ax5000ParamSTRUCTs/P/AX5000_P_0901
TYPE AX5000_P_0901 :
STRUCT
	Safe_factory_settings:UINT;
END_STRUCT
END_TYPE

// POUs/IO/Drives/SoE/Ax5000ParamSTRUCTs/P/AX5000_P_0902
TYPE AX5000_P_0902 :
STRUCT
	Current_calibration:UINT;
END_STRUCT
END_TYPE

// POUs/IO/Drives/SoE/Ax5000ParamSTRUCTs/P/AX5000_P_0904
TYPE AX5000_P_0904 :
STRUCT
	Save_device_component_hardware_Ids:UINT;
END_STRUCT
END_TYPE

// POUs/IO/Drives/SoE/Ax5000ParamSTRUCTs/P/AX5000_P_0905
TYPE AX5000_P_0905 :
STRUCT
	Clear_error_history:UINT;
END_STRUCT
END_TYPE

// POUs/IO/Drives/SoE/Ax5000ParamSTRUCTs/P/AX5000_P_0906
TYPE AX5000_P_0906 :
STRUCT
	Reset_operation_times:UINT;
END_STRUCT
END_TYPE

// POUs/IO/Drives/SoE/Ax5000ParamSTRUCTs/P/AX5000_P_0912
TYPE AX5000_P_0912 :
STRUCT
	Actual_lenght:UINT;
	Max_lenght:UINT;
	Calibration:UINT;
	Calibration_type:UINT;
	Calibration_point:UINT;
	Calibration_current:UINT;
	Calibration_phase:UINT;
	Calibration_tolerance:UINT;
END_STRUCT
END_TYPE

// POUs/IO/Drives/SoE/Ax5000ParamSTRUCTs/P/AX5000_P_1000
TYPE AX5000_P_1000 :
STRUCT
	Debug_pointer_1_adr:UDINT;
END_STRUCT
END_TYPE

// POUs/IO/Drives/SoE/Ax5000ParamSTRUCTs/P/AX5000_P_1001
TYPE AX5000_P_1001 :
STRUCT
	Debug_pointer_1_typ:UINT;
END_STRUCT
END_TYPE

// POUs/IO/Drives/SoE/Ax5000ParamSTRUCTs/P/AX5000_P_1002
TYPE AX5000_P_1002 :
STRUCT
	Debug_pointer_1_value:UDINT;
END_STRUCT
END_TYPE

// POUs/IO/Drives/SoE/Ax5000ParamSTRUCTs/P/AX5000_P_1003
TYPE AX5000_P_1003 :
STRUCT
	Debug_pointer_2_adr:UDINT;
END_STRUCT
END_TYPE

// POUs/IO/Drives/SoE/Ax5000ParamSTRUCTs/P/AX5000_P_1004
TYPE AX5000_P_1004 :
STRUCT
	Debug_pointer_2_type:UINT;
END_STRUCT
END_TYPE

// POUs/IO/Drives/SoE/Ax5000ParamSTRUCTs/P/AX5000_P_1005
TYPE AX5000_P_1005 :
STRUCT
	Debug_pointer_2_value:UDINT;
END_STRUCT
END_TYPE

// POUs/IO/Drives/SoE/Ax5000ParamSTRUCTs/P/AX5000_P_1006
TYPE AX5000_P_1006 :
STRUCT
	Addr:UINT;
	Source:UINT;
END_STRUCT
END_TYPE

// POUs/IO/Drives/SoE/Ax5000ParamSTRUCTs/P/AX5000_P_1007
TYPE AX5000_P_1007 :
STRUCT
	Feedback_debug_pointer_1_typ:UINT;
END_STRUCT
END_TYPE

// POUs/IO/Drives/SoE/Ax5000ParamSTRUCTs/P/AX5000_P_1008
TYPE AX5000_P_1008 :
STRUCT
	Feedback_debug_pointer_1_value:UINT;
END_STRUCT
END_TYPE

// POUs/IO/Drives/SoE/Ax5000ParamSTRUCTs/P/AX5000_P_1009
TYPE AX5000_P_1009 :
STRUCT
	Addr:UINT;
	Source:UINT;
END_STRUCT
END_TYPE

// POUs/IO/Drives/SoE/Ax5000ParamSTRUCTs/P/AX5000_P_1010
TYPE AX5000_P_1010 :
STRUCT
	Feedback_debug_pointer_2_vtype:UINT;
END_STRUCT
END_TYPE

// POUs/IO/Drives/SoE/Ax5000ParamSTRUCTs/P/AX5000_P_1011
TYPE AX5000_P_1011 :
STRUCT
	Feedback_debug_pointer_2_value:UINT;
END_STRUCT
END_TYPE

// POUs/IO/Drives/SoE/Ax5000ParamSTRUCTs/P/AX5000_P_1012
TYPE AX5000_P_1012 :
STRUCT
	Memory_dump_selector:UINT;
END_STRUCT
END_TYPE

// POUs/IO/Drives/SoE/Ax5000ParamSTRUCTs/P/AX5000_P_1020
TYPE AX5000_P_1020 :
STRUCT
	Debug_parameter:UINT;
END_STRUCT
END_TYPE

// POUs/IO/Drives/SoE/Ax5000ParamSTRUCTs/P/AX5000_P_1021
TYPE AX5000_P_1021 :
STRUCT
	Debug_variable:UDINT;
END_STRUCT
END_TYPE

// POUs/IO/Drives/SoE/Ax5000ParamSTRUCTs/P/AX5000_P_1022
TYPE AX5000_P_1022 :
STRUCT
	Deburg_command:UINT;
END_STRUCT
END_TYPE

// POUs/IO/Drives/SoE/Ax5000ParamSTRUCTs/P/AX5000_P_2000
TYPE AX5000_P_2000 :
STRUCT
	Configured_safety_option: E_AX5000_P_2000_SafetyOption;
END_STRUCT
END_TYPE

// POUs/IO/Drives/SoE/Ax5000ParamSTRUCTs/P/AX5000_P_2001
TYPE AX5000_P_2001 :
STRUCT
	Safety_option_diagnostics:UINT;
END_STRUCT
END_TYPE

// POUs/IO/Drives/SoE/Ax5000ParamSTRUCTs/P/AX5000_P_2002
TYPE AX5000_P_2002 :
STRUCT
	Safety_option_state:UINT;
END_STRUCT
END_TYPE

// POUs/IO/Drives/SoE/Ax5000ParamSTRUCTs/S/AX5000_S_0001
TYPE AX5000_S_0001 :
STRUCT
	Switching_frequency_of_the_IGBT_module:UINT;
END_STRUCT
END_TYPE

// POUs/IO/Drives/SoE/Ax5000ParamSTRUCTs/S/AX5000_S_0002
TYPE AX5000_S_0002 :
STRUCT
	Communication_cycle_time:UINT;
END_STRUCT
END_TYPE

// POUs/IO/Drives/SoE/Ax5000ParamSTRUCTs/S/AX5000_S_0007
TYPE AX5000_S_0007 :
STRUCT
	Feedvack_acquisition_capture_point:UINT;
END_STRUCT
END_TYPE

// POUs/IO/Drives/SoE/Ax5000ParamSTRUCTs/S/AX5000_S_0011
TYPE AX5000_S_0011 :
STRUCT
	Class_1_diagnostic:UINT;
END_STRUCT
END_TYPE

// POUs/IO/Drives/SoE/Ax5000ParamSTRUCTs/S/AX5000_S_0012
TYPE AX5000_S_0012 :
STRUCT
	Class_2_diagnostic:UINT;
END_STRUCT
END_TYPE

// POUs/IO/Drives/SoE/Ax5000ParamSTRUCTs/S/AX5000_S_0013
TYPE AX5000_S_0013 :
STRUCT
	Class_3_diagnostic:UINT;
END_STRUCT
END_TYPE

// POUs/IO/Drives/SoE/Ax5000ParamSTRUCTs/S/AX5000_S_0015
TYPE AX5000_S_0015 :
STRUCT
	Telefram_type:UINT;
END_STRUCT
END_TYPE

// POUs/IO/Drives/SoE/Ax5000ParamSTRUCTs/S/AX5000_S_0016
TYPE AX5000_S_0016 :
STRUCT
	Actual_lenght:UINT;
	Max_lenght:UINT;
	Configuration_list_of_AT:ARRAY[0..23] OF UINT;
END_STRUCT
END_TYPE

// POUs/IO/Drives/SoE/Ax5000ParamSTRUCTs/S/AX5000_S_0017
TYPE AX5000_S_0017 :
STRUCT
	Actual_lenght:UINT;
	Max_lenght:UINT;
	IDN_list_of_all_operation_data: ARRAY[0..693] OF UINT;
END_STRUCT
END_TYPE

// POUs/IO/Drives/SoE/Ax5000ParamSTRUCTs/S/AX5000_S_0018
TYPE AX5000_S_0018 :
STRUCT
	Actual_lenght:UINT;
	Max_lenght:UINT;
	IDN_list_of_all_operation_data_for_CP2: ARRAY[0..346] OF UINT;
END_STRUCT
END_TYPE

// POUs/IO/Drives/SoE/Ax5000ParamSTRUCTs/S/AX5000_S_0024
TYPE AX5000_S_0024 :
STRUCT
	Actual_lenght:UINT;
	Max_lenght:UINT;
	Configuration_list_of_MDT:ARRAY[0..11] OF UINT;
END_STRUCT
END_TYPE

// POUs/IO/Drives/SoE/Ax5000ParamSTRUCTs/S/AX5000_S_0029
TYPE AX5000_S_0029 :
STRUCT
	MDT_error_counter:UINT;
END_STRUCT
END_TYPE

// POUs/IO/Drives/SoE/Ax5000ParamSTRUCTs/S/AX5000_S_0030
TYPE AX5000_S_0030 :
STRUCT
	Actual_lenght:UINT;
	Max_lenght:UINT;
	Manufacturer_version:STRING(61);
END_STRUCT
END_TYPE

// POUs/IO/Drives/SoE/Ax5000ParamSTRUCTs/S/AX5000_S_0031
TYPE AX5000_S_0031 :
STRUCT
	Actual_lenght:UINT;
	Max_lenght:UINT;
	Hardware_version:STRING(45)
;END_STRUCT
END_TYPE

// POUs/IO/Drives/SoE/Ax5000ParamSTRUCTs/S/AX5000_S_0032
TYPE AX5000_S_0032 :
STRUCT
	Primary_operation_mode:E_AX5000_S_0032_OperationMode;
END_STRUCT
END_TYPE

// POUs/IO/Drives/SoE/Ax5000ParamSTRUCTs/S/AX5000_S_0033
TYPE AX5000_S_0033 :
STRUCT
	Secondary_operation_mode1:UINT;
END_STRUCT
END_TYPE

// POUs/IO/Drives/SoE/Ax5000ParamSTRUCTs/S/AX5000_S_0034
TYPE AX5000_S_0034 :
STRUCT
	Secondary_operation_mode2:UINT;
END_STRUCT
END_TYPE

// POUs/IO/Drives/SoE/Ax5000ParamSTRUCTs/S/AX5000_S_0035
TYPE AX5000_S_0035 :
STRUCT
	Secondary_operation_mode3:UINT;
END_STRUCT
END_TYPE

// POUs/IO/Drives/SoE/Ax5000ParamSTRUCTs/S/AX5000_S_0036
TYPE AX5000_S_0036 :
STRUCT
	Velocity_command_value:DINT;
END_STRUCT
END_TYPE

// POUs/IO/Drives/SoE/Ax5000ParamSTRUCTs/S/AX5000_S_0037
TYPE AX5000_S_0037 :
STRUCT
	Additive_Velocity_command_value:DINT;
END_STRUCT
END_TYPE

// POUs/IO/Drives/SoE/Ax5000ParamSTRUCTs/S/AX5000_S_0040
TYPE AX5000_S_0040 :
STRUCT
	Velocity_feedback_value1:DINT;
END_STRUCT
END_TYPE

// POUs/IO/Drives/SoE/Ax5000ParamSTRUCTs/S/AX5000_S_0043
TYPE AX5000_S_0043 :
STRUCT
	Velocity_polarity_parameter:UINT;
END_STRUCT
END_TYPE

// POUs/IO/Drives/SoE/Ax5000ParamSTRUCTs/S/AX5000_S_0044
TYPE AX5000_S_0044 :
STRUCT
	Velocity_data_scaling_type:UINT;
END_STRUCT
END_TYPE

// POUs/IO/Drives/SoE/Ax5000ParamSTRUCTs/S/AX5000_S_0045
TYPE AX5000_S_0045 :
STRUCT
	Velocity_data_scaling_factor:UINT;
END_STRUCT
END_TYPE

// POUs/IO/Drives/SoE/Ax5000ParamSTRUCTs/S/AX5000_S_0046
TYPE AX5000_S_0046 :
STRUCT
	Velocity_data_scaling_exponent:INT;
END_STRUCT
END_TYPE

// POUs/IO/Drives/SoE/Ax5000ParamSTRUCTs/S/AX5000_S_0047
TYPE AX5000_S_0047 :
STRUCT
	Position_command_valut:DINT;
END_STRUCT
END_TYPE

// POUs/IO/Drives/SoE/Ax5000ParamSTRUCTs/S/AX5000_S_0048
TYPE AX5000_S_0048 :
STRUCT
	Additive_position_command_value:DINT;
END_STRUCT
END_TYPE

// POUs/IO/Drives/SoE/Ax5000ParamSTRUCTs/S/AX5000_S_0051
TYPE AX5000_S_0051 :
STRUCT
	Position_feedback_value_1:DINT;
END_STRUCT
END_TYPE

// POUs/IO/Drives/SoE/Ax5000ParamSTRUCTs/S/AX5000_S_0053
TYPE AX5000_S_0053 :
STRUCT
	Position_feedback_value_2:DINT;
END_STRUCT
END_TYPE

// POUs/IO/Drives/SoE/Ax5000ParamSTRUCTs/S/AX5000_S_0055
TYPE AX5000_S_0055 :
STRUCT
	Position_polatity_parameter:UINT;
END_STRUCT
END_TYPE

// POUs/IO/Drives/SoE/Ax5000ParamSTRUCTs/S/AX5000_S_0076
TYPE AX5000_S_0076 EXTENDS ST_AX5000_S_0076:
STRUCT
//	Position_data_scaling_type:UINT;
END_STRUCT
END_TYPE

// POUs/IO/Drives/SoE/Ax5000ParamSTRUCTs/S/AX5000_S_0079
TYPE AX5000_S_0079 :
STRUCT
	Rotational_position_resolution:UDINT;
END_STRUCT
END_TYPE

// POUs/IO/Drives/SoE/Ax5000ParamSTRUCTs/S/AX5000_S_0080
TYPE AX5000_S_0080 :
STRUCT
	Torque_command_value:INT;
END_STRUCT
END_TYPE

// POUs/IO/Drives/SoE/Ax5000ParamSTRUCTs/S/AX5000_S_0081
TYPE AX5000_S_0081 :
STRUCT
	Additive_Torque_command_value:INT;
END_STRUCT
END_TYPE

// POUs/IO/Drives/SoE/Ax5000ParamSTRUCTs/S/AX5000_S_0082
TYPE AX5000_S_0082 :
STRUCT
	Positiv_Torque_command_value:UINT;
END_STRUCT
END_TYPE

// POUs/IO/Drives/SoE/Ax5000ParamSTRUCTs/S/AX5000_S_0083
TYPE AX5000_S_0083 :
STRUCT
	Negative_Torque_command_value:UINT;
END_STRUCT
END_TYPE

// POUs/IO/Drives/SoE/Ax5000ParamSTRUCTs/S/AX5000_S_0084
TYPE AX5000_S_0084 :
STRUCT
	Torque_feedback_value:INT;
END_STRUCT
END_TYPE

// POUs/IO/Drives/SoE/Ax5000ParamSTRUCTs/S/AX5000_S_0085
TYPE AX5000_S_0085 EXTENDS ST_AX5000_S_0085:
STRUCT
//	Torque_polarity_parameter:UINT;
END_STRUCT
END_TYPE

// POUs/IO/Drives/SoE/Ax5000ParamSTRUCTs/S/AX5000_S_0086
TYPE AX5000_S_0086 :
STRUCT
	Torque_force_data_scaling_type:UINT;
END_STRUCT
END_TYPE

// POUs/IO/Drives/SoE/Ax5000ParamSTRUCTs/S/AX5000_S_0091
TYPE AX5000_S_0091 :
STRUCT
	Bipolar_velocity_limit_value:UDINT;
END_STRUCT
END_TYPE

// POUs/IO/Drives/SoE/Ax5000ParamSTRUCTs/S/AX5000_S_0092
TYPE AX5000_S_0092 :
STRUCT
	Bipolar_torqu_limit_value:UINT;
END_STRUCT
END_TYPE

// POUs/IO/Drives/SoE/Ax5000ParamSTRUCTs/S/AX5000_S_0095
TYPE AX5000_S_0095 :
STRUCT
	Actual_lenght:UINT;
	Max_lenght:UINT;
	Diagnistic_message:STRING(99);
END_STRUCT
END_TYPE

// POUs/IO/Drives/SoE/Ax5000ParamSTRUCTs/S/AX5000_S_0099
TYPE AX5000_S_0099 :
STRUCT
	Reset_class_1_diagnistic:UINT;
END_STRUCT
END_TYPE

// POUs/IO/Drives/SoE/Ax5000ParamSTRUCTs/S/AX5000_S_0100
TYPE AX5000_S_0100 :
STRUCT
	Velocity_loop_proportional_gain:UDINT;
END_STRUCT
END_TYPE

// POUs/IO/Drives/SoE/Ax5000ParamSTRUCTs/S/AX5000_S_0101
TYPE AX5000_S_0101 :
STRUCT
	Velocity_loop_integral_action_time:UINT;
END_STRUCT
END_TYPE

// POUs/IO/Drives/SoE/Ax5000ParamSTRUCTs/S/AX5000_S_0103
TYPE AX5000_S_0103 :
STRUCT
	Moduo_value:UDINT;
END_STRUCT
END_TYPE

// POUs/IO/Drives/SoE/Ax5000ParamSTRUCTs/S/AX5000_S_0104
TYPE AX5000_S_0104 :
STRUCT
	Position_loop_Kv_factor:UINT;
END_STRUCT
END_TYPE

// POUs/IO/Drives/SoE/Ax5000ParamSTRUCTs/S/AX5000_S_0106
TYPE AX5000_S_0106 :
STRUCT
	Current_loop_proportional_gain_1:UINT;
END_STRUCT
END_TYPE

// POUs/IO/Drives/SoE/Ax5000ParamSTRUCTs/S/AX5000_S_0107
TYPE AX5000_S_0107 :
STRUCT
	Current_conrol_loop_integral_action_time1:UINT;
END_STRUCT
END_TYPE

// POUs/IO/Drives/SoE/Ax5000ParamSTRUCTs/S/AX5000_S_0109
TYPE AX5000_S_0109 :
STRUCT
	Motor_peak_current:UDINT;
END_STRUCT
END_TYPE

// POUs/IO/Drives/SoE/Ax5000ParamSTRUCTs/S/AX5000_S_0110
TYPE AX5000_S_0110 :
STRUCT
	Amplifier_peak_current:UDINT;
END_STRUCT
END_TYPE

// POUs/IO/Drives/SoE/Ax5000ParamSTRUCTs/S/AX5000_S_0111
TYPE AX5000_S_0111 :
STRUCT
	Motor_continouse_stall_current:UINT;
END_STRUCT
END_TYPE

// POUs/IO/Drives/SoE/Ax5000ParamSTRUCTs/S/AX5000_S_0112
TYPE AX5000_S_0112 :
STRUCT
	Amplifier_rated_current:UDINT;
END_STRUCT
END_TYPE

// POUs/IO/Drives/SoE/Ax5000ParamSTRUCTs/S/AX5000_S_0113
TYPE AX5000_S_0113 :
STRUCT
	Maximum_motor_speed:UDINT;
END_STRUCT
END_TYPE

// POUs/IO/Drives/SoE/Ax5000ParamSTRUCTs/S/AX5000_S_0119
TYPE AX5000_S_0119 :
STRUCT
	Current_loop_proportional_gain2:UINT;
END_STRUCT
END_TYPE

// POUs/IO/Drives/SoE/Ax5000ParamSTRUCTs/S/AX5000_S_0120
TYPE AX5000_S_0120 :
STRUCT
	Current_controler_loop_integral_action_time2:UINT;
END_STRUCT
END_TYPE

// POUs/IO/Drives/SoE/Ax5000ParamSTRUCTs/S/AX5000_S_0124
TYPE AX5000_S_0124 :
STRUCT
	Standstill_window:UDINT;
END_STRUCT
END_TYPE

// POUs/IO/Drives/SoE/Ax5000ParamSTRUCTs/S/AX5000_S_0126
TYPE AX5000_S_0126 :
STRUCT
	Torque_threshold_Tx:UINT;
END_STRUCT
END_TYPE

// POUs/IO/Drives/SoE/Ax5000ParamSTRUCTs/S/AX5000_S_0130
TYPE AX5000_S_0130 :
STRUCT
	Probe_value_1_positive_edge:DINT;
END_STRUCT
END_TYPE

// POUs/IO/Drives/SoE/Ax5000ParamSTRUCTs/S/AX5000_S_0131
TYPE AX5000_S_0131 :
STRUCT
	Probe_value_1_negative_edge:DINT;
END_STRUCT
END_TYPE

// POUs/IO/Drives/SoE/Ax5000ParamSTRUCTs/S/AX5000_S_0134
TYPE AX5000_S_0134 :
STRUCT
	Master_controll_word:UINT;
END_STRUCT
END_TYPE

// POUs/IO/Drives/SoE/Ax5000ParamSTRUCTs/S/AX5000_S_0135
TYPE AX5000_S_0135 :
STRUCT
	Drive_status_word:UINT;
END_STRUCT
END_TYPE

// POUs/IO/Drives/SoE/Ax5000ParamSTRUCTs/S/AX5000_S_0136
TYPE AX5000_S_0136 :
STRUCT
	Positive_acceleration_limit_value:UDINT;
END_STRUCT
END_TYPE

// POUs/IO/Drives/SoE/Ax5000ParamSTRUCTs/S/AX5000_S_0137
TYPE AX5000_S_0137 :
STRUCT
	Negative_acceleration_limit_value:UDINT;
END_STRUCT
END_TYPE

// POUs/IO/Drives/SoE/Ax5000ParamSTRUCTs/S/AX5000_S_0143
TYPE AX5000_S_0143 :
STRUCT
	Actual_lenght:UINT;
	Max_lenght:UINT;
	Sercos_interface_version:STRING(8);
END_STRUCT
END_TYPE

// POUs/IO/Drives/SoE/Ax5000ParamSTRUCTs/S/AX5000_S_0149
TYPE AX5000_S_0149 :
STRUCT
	Positive_drive_stop_procedure_command:UINT;
END_STRUCT
END_TYPE

// POUs/IO/Drives/SoE/Ax5000ParamSTRUCTs/S/AX5000_S_0159
TYPE AX5000_S_0159 :
STRUCT
	Monitoring_window:UDINT;
END_STRUCT
END_TYPE

// POUs/IO/Drives/SoE/Ax5000ParamSTRUCTs/S/AX5000_S_0160
TYPE AX5000_S_0160 :
STRUCT
	Acceleration_data_scaling_type:UINT;
END_STRUCT
END_TYPE

// POUs/IO/Drives/SoE/Ax5000ParamSTRUCTs/S/AX5000_S_0161
TYPE AX5000_S_0161 :
STRUCT
	Acceleration_data_scaling_factor:UINT;
END_STRUCT
END_TYPE

// POUs/IO/Drives/SoE/Ax5000ParamSTRUCTs/S/AX5000_S_0162
TYPE AX5000_S_0162 :
STRUCT
	Acceleration_data_scaling_exponent:UINT;
END_STRUCT
END_TYPE

// POUs/IO/Drives/SoE/Ax5000ParamSTRUCTs/S/AX5000_S_0163
TYPE AX5000_S_0163 :
STRUCT
	Weight_counterbalance:INT;
END_STRUCT
END_TYPE

// POUs/IO/Drives/SoE/Ax5000ParamSTRUCTs/S/AX5000_S_0169
TYPE AX5000_S_0169 :
STRUCT
//	Probe_control_parameter:UINT;
	
(* 0=Not Active, 1=Active *)
		Probe1PositiveEdge : BIT;
		(* 0=Not Active, 1=Active *)
		Probe1NegativeEdge : BIT;
		 {attribute 'hide'}
		_reserved1 : BIT;
		 {attribute 'hide'}
		_reserved2 : BIT;
		 {attribute 'hide'}
		_reserved3 : BIT;
		(* 0=Single Measuring, 1=Continous Measuring *)
		ModeProbe1 : BIT;
		 {attribute 'hide'}
		_reserved4 : BIT;
		 {attribute 'hide'}
		_reserved5 : BIT;
		(* 0=Ativation with S170, 1=Autoactivation from SafeOp to Op *)
		AutoActivation : BIT;
		 {attribute 'hide'}
		_reserved6 : BIT;
		 {attribute 'hide'}
		_reserved7 : BIT;
		 {attribute 'hide'}
		_reserved8 : BIT;
		 {attribute 'hide'}
		_reserved9 : BIT;
		 {attribute 'hide'}
		_reserved10 : BIT;
		 {attribute 'hide'}
		_reserved11 : BIT;
		 {attribute 'hide'}
		_reserved12 : BIT;
END_STRUCT
END_TYPE

// POUs/IO/Drives/SoE/Ax5000ParamSTRUCTs/S/AX5000_S_0170
TYPE AX5000_S_0170 :
STRUCT
	Probing_cycle_procedure_command:UINT;
END_STRUCT
END_TYPE

// POUs/IO/Drives/SoE/Ax5000ParamSTRUCTs/S/AX5000_S_0179
TYPE AX5000_S_0179 :
STRUCT
	Probe_status:UINT;
END_STRUCT
END_TYPE

// POUs/IO/Drives/SoE/Ax5000ParamSTRUCTs/S/AX5000_S_0185
TYPE AX5000_S_0185 :
STRUCT
	Length_of_the_configurabel_data_record_in_the_AT:UINT;
END_STRUCT
END_TYPE

// POUs/IO/Drives/SoE/Ax5000ParamSTRUCTs/S/AX5000_S_0186
TYPE AX5000_S_0186 :
STRUCT
	Length_of_the_configurabel_data_record_in_the_MDT:UINT;
END_STRUCT
END_TYPE

// POUs/IO/Drives/SoE/Ax5000ParamSTRUCTs/S/AX5000_S_0187
TYPE AX5000_S_0187 :
STRUCT
	Actual_lenght:UINT;
	Max_lenght:UINT;
	IDN_list_of_configurable_data_in_the_AT:ARRAY[0..67] OF UINT;
END_STRUCT
END_TYPE

// POUs/IO/Drives/SoE/Ax5000ParamSTRUCTs/S/AX5000_S_0188
TYPE AX5000_S_0188 :
STRUCT
	Actual_lenght:UINT;
	Max_lenght:UINT;
	IDN_list_of_configurable_data_in_the_AT:ARRAY[0..13] OF UINT;
END_STRUCT
END_TYPE

// POUs/IO/Drives/SoE/Ax5000ParamSTRUCTs/S/AX5000_S_0189
TYPE AX5000_S_0189 :
STRUCT
	following_distance:DINT;
END_STRUCT
END_TYPE

// POUs/IO/Drives/SoE/Ax5000ParamSTRUCTs/S/AX5000_S_0196
TYPE AX5000_S_0196 :
STRUCT
	Motor_rated_current:UDINT;
END_STRUCT
END_TYPE

// POUs/IO/Drives/SoE/Ax5000ParamSTRUCTs/S/AX5000_S_0200
TYPE AX5000_S_0200 :
STRUCT
	Amplifier_warning_temperature:UINT;
END_STRUCT
END_TYPE

// POUs/IO/Drives/SoE/Ax5000ParamSTRUCTs/S/AX5000_S_0201
TYPE AX5000_S_0201 :
STRUCT
	Motor_warning_temperature:UINT;
END_STRUCT
END_TYPE

// POUs/IO/Drives/SoE/Ax5000ParamSTRUCTs/S/AX5000_S_0203
TYPE AX5000_S_0203 :
STRUCT
	Amplifier_shut_down_temperature:UINT;
END_STRUCT
END_TYPE

// POUs/IO/Drives/SoE/Ax5000ParamSTRUCTs/S/AX5000_S_0204
TYPE AX5000_S_0204 :
STRUCT
	Motor_shut_down_temperature:UINT;
END_STRUCT
END_TYPE

// POUs/IO/Drives/SoE/Ax5000ParamSTRUCTs/S/AX5000_S_0206
TYPE AX5000_S_0206 :
STRUCT
	Drive_of_delay_time:UINT;
END_STRUCT
END_TYPE

// POUs/IO/Drives/SoE/Ax5000ParamSTRUCTs/S/AX5000_S_0207
TYPE AX5000_S_0207 :
STRUCT
	Drive_delay_time:UINT;
END_STRUCT
END_TYPE

// POUs/IO/Drives/SoE/Ax5000ParamSTRUCTs/S/AX5000_S_0216
TYPE AX5000_S_0216 :
STRUCT
	Switch_parameter:UINT;
END_STRUCT
END_TYPE

// POUs/IO/Drives/SoE/Ax5000ParamSTRUCTs/S/AX5000_S_0217
TYPE AX5000_S_0217 :
STRUCT
	Parameter_set_preselection:UINT;
END_STRUCT
END_TYPE

// POUs/IO/Drives/SoE/Ax5000ParamSTRUCTs/S/AX5000_S_0219
TYPE AX5000_S_0219 :
STRUCT
	Actual_lenght:UINT;
	Max_lenght:UINT;
	IDN_list_of_parameter_set:ARRAY[0..44] OF UINT;
END_STRUCT
END_TYPE

// POUs/IO/Drives/SoE/Ax5000ParamSTRUCTs/S/AX5000_S_0254
TYPE AX5000_S_0254 :
STRUCT
	Actual_parameter_set:UINT;
END_STRUCT
END_TYPE

// POUs/IO/Drives/SoE/Ax5000ParamSTRUCTs/S/AX5000_S_0256
TYPE AX5000_S_0256 :
STRUCT
	Multiplication_factor1:UDINT;
END_STRUCT
END_TYPE

// POUs/IO/Drives/SoE/Ax5000ParamSTRUCTs/S/AX5000_S_0257
TYPE AX5000_S_0257 :
STRUCT
	Multiplication_factor2:UDINT;
END_STRUCT
END_TYPE

// POUs/IO/Drives/SoE/Ax5000ParamSTRUCTs/S/AX5000_S_0267
TYPE AX5000_S_0267 :
STRUCT
	Actual_lenght:UINT;
	Max_lenght:UINT;
	Password:STRING(29);
END_STRUCT
END_TYPE

// POUs/IO/Drives/SoE/Ax5000ParamSTRUCTs/S/AX5000_S_0273
TYPE AX5000_S_0273 :
STRUCT
	Maximum_drive_off_delay_time:UDINT;
END_STRUCT
END_TYPE

// POUs/IO/Drives/SoE/Ax5000ParamSTRUCTs/S/AX5000_S_0274
TYPE AX5000_S_0274 :
STRUCT
	Actual_lenght:UINT;
	Max_lenght:UINT;
	Received_drive_addresses:UINT;
END_STRUCT
END_TYPE

// POUs/IO/Drives/SoE/Ax5000ParamSTRUCTs/S/AX5000_S_0292
TYPE AX5000_S_0292 :
STRUCT
	Actual_lenght:UINT;
	Max_lenght:UINT;
	List_of_supported_operation_modes: ARRAY[0..5] OF UINT;
END_STRUCT
END_TYPE

// POUs/IO/Drives/SoE/Ax5000ParamSTRUCTs/S/AX5000_S_0295
TYPE AX5000_S_0295 :
STRUCT
	Drive_enable_delay_time:UINT;
END_STRUCT
END_TYPE

// POUs/IO/Drives/SoE/Ax5000ParamSTRUCTs/S/AX5000_S_0296
TYPE AX5000_S_0296 :
STRUCT
	Velocity_feed_forword_gain:UINT;
END_STRUCT
END_TYPE

// POUs/IO/Drives/SoE/Ax5000ParamSTRUCTs/S/AX5000_S_0347
TYPE AX5000_S_0347 :
STRUCT
	Velocity_error:DINT;
END_STRUCT
END_TYPE

// POUs/IO/Drives/SoE/Ax5000ParamSTRUCTs/S/AX5000_S_0348
TYPE AX5000_S_0348 :
STRUCT
	Acceleration_feed_forword_gain:UINT;
END_STRUCT
END_TYPE

// POUs/IO/Drives/SoE/Ax5000ParamSTRUCTs/S/AX5000_S_0372
TYPE AX5000_S_0372 :
STRUCT
	Drive_Halt_acceleration_bipolar:DINT;
END_STRUCT
END_TYPE

// POUs/IO/Drives/SoE/Ax5000ParamSTRUCTs/S/AX5000_S_0374
TYPE AX5000_S_0374 :
STRUCT
	Actual_lenght:UINT;
	Max_lenght:UINT;
	Procedure_command_error_list:ARRAY[0..59] OF UINT;
END_STRUCT
END_TYPE

// POUs/IO/Drives/SoE/Ax5000ParamSTRUCTs/S/AX5000_S_0375
TYPE AX5000_S_0375 :
STRUCT
	Actual_lenght:UINT;
	Max_lenght:UINT;
	Diagnostic_number_list:ARRAY[0..59] OF UINT;
END_STRUCT
END_TYPE

// POUs/IO/Drives/SoE/Ax5000ParamSTRUCTs/S/AX5000_S_0380
TYPE AX5000_S_0380 :
STRUCT
	DC_bus_voltage:UINT;
END_STRUCT
END_TYPE

// POUs/IO/Drives/SoE/Ax5000ParamSTRUCTs/S/AX5000_S_0381
TYPE AX5000_S_0381 :
STRUCT
	DC_bus_current:DINT;
END_STRUCT
END_TYPE

// POUs/IO/Drives/SoE/Ax5000ParamSTRUCTs/S/AX5000_S_0383
TYPE AX5000_S_0383 :
STRUCT
	Motor_temperature:UINT;
END_STRUCT
END_TYPE

// POUs/IO/Drives/SoE/Ax5000ParamSTRUCTs/S/AX5000_S_0384
TYPE AX5000_S_0384 :
STRUCT
	Amplifier_temperature:UINT;
END_STRUCT
END_TYPE

// POUs/IO/Drives/SoE/Ax5000ParamSTRUCTs/S/AX5000_S_0390
TYPE AX5000_S_0390 :
STRUCT
	Diagnostic_number:UDINT;
END_STRUCT
END_TYPE

// POUs/IO/Drives/SoE/Ax5000ParamSTRUCTs/S/AX5000_S_0403
TYPE AX5000_S_0403 :
STRUCT
	Position_feedback_value_status:UINT;
END_STRUCT
END_TYPE

// POUs/IO/Drives/SoE/Ax5000ParamSTRUCTs/S/AX5000_S_0405
TYPE AX5000_S_0405 :
STRUCT
	Probe1_enable:UINT;
END_STRUCT
END_TYPE

// POUs/IO/Drives/SoE/Ax5000ParamSTRUCTs/S/AX5000_S_0409
TYPE AX5000_S_0409 :
STRUCT
	Probe1_positive_latched:UINT;
END_STRUCT
END_TYPE

// POUs/IO/Drives/SoE/Ax5000ParamSTRUCTs/S/AX5000_S_0410
TYPE AX5000_S_0410 :
STRUCT
	Probe1_negative_latched:UINT;
END_STRUCT
END_TYPE

// POUs/IO/Drives/SoE/Ax5000ParamSTRUCTs/S/AX5000_S_0429
TYPE AX5000_S_0429 :
STRUCT
	Emergancey_stop_decleration:UDINT;
END_STRUCT
END_TYPE

// POUs/IO/Drives/SoE/Ax5000ParamSTRUCTs/S/AX5000_S_0432
TYPE AX5000_S_0432 :
STRUCT
	Actual_lenght:UINT;
	Max_lenght:UINT;
	Serial_number_drive_control:STRING(18);
END_STRUCT
END_TYPE

// POUs/IO/Drives/SoE/Ax5000ParamSTRUCTs/S/AX5000_S_0435
TYPE AX5000_S_0435 :
STRUCT
	Operating_time_drive_control:UDINT;
END_STRUCT
END_TYPE

// POUs/IO/Drives/SoE/Ax5000ParamSTRUCTs/S/AX5000_S_0436
TYPE AX5000_S_0436 :
STRUCT
	Operating_time_power_stage:UDINT;
END_STRUCT
END_TYPE

// POUs/Logging/LogbookData
TYPE LogbookData :
STRUCT
	Timestamp												:	TIMESTRUCT;						//Stored timestamp for each message
	Msg														:	STRING(PARAM.LOGBOOK_MAX_MSG_STRING_LENGHT); //Stored message
{attribute 'displaymode':='binary'}	
	Options													:	WORD;							//Stored option for each message
END_STRUCT
END_TYPE

// POUs/Motion/TF511x-KIN/03_DUTs/Positions/KIN_POSITIONS_ACS_DUT
TYPE KIN_POSITIONS_ACS_DUT :
STRUCT
	A1					: LREAL; //Joint axis 1
	A2					: LREAL; //Joint axis 2
	A3					: LREAL; //Joint axis 3
	A4					: LREAL; //Joint axis 4
	A5					: LREAL; //Joint axis 5
	A6					: LREAL; //Joint axis 6
	Q1					: LREAL; //Auxiliary joint axis 1
	Q2					: LREAL; //Auxiliary joint axis 2 	
END_STRUCT
END_TYPE

// POUs/Motion/TF511x-KIN/03_DUTs/Positions/KIN_POSITIONS_MCS_DUT
TYPE KIN_POSITIONS_MCS_DUT EXTENDS VALUE_6D_DUT:
STRUCT
	Q1					: LREAL; //Auxiliary axis 1
	Q2					: LREAL; //Auxiliary axis 2 	
END_STRUCT
END_TYPE

// POUs/Motion/TF511x-KIN/03_DUTs/Positions/U_KIN_POSITIONS
TYPE U_KIN_POSITIONS :  //Union datatype for kinematic positions in different identifier
UNION
	MCS							:	KIN_POSITIONS_MCS_DUT; //XYZ ABC Q1,Q2
	ACS							:	KIN_POSITIONS_ACS_DUT; //A1..A6,Q1,Q2
	Joints						:	ARRAY[1..8] OF LREAL; //Array 1..8
END_UNION
END_TYPE

// POUs/Motion/VALUE_3D_DUT
TYPE VALUE_3D_DUT :
STRUCT
	X					:		LREAL;
	Y					:		LREAL;
	Z					:		LREAL;
END_STRUCT
END_TYPE

// POUs/Motion/VALUE_6D_DUT
TYPE VALUE_6D_DUT EXTENDS VALUE_3D_DUT:
STRUCT
	A					:		LREAL; //Rx
	B					:		LREAL; //Ry
	C					:		LREAL; //Rz	
END_STRUCT
END_TYPE

// POUs/Safety/SAFETY_CIRCUIT_STATUS
TYPE SAFETY_CIRCUIT_STATUS :
STRUCT
	State													:	eSTATE := eSTATE.ABORTED;

	InAborting												:	BOOL; //MonOut switched to false, MonDelOut still true
	InAborted												:	BOOL; //MonOut and MonDelOut = FALSE
	InClearing												:	BOOL; //MonOut and MonDelOut = TRUE, OK delay time is running
	InIdle													:	BOOL; //OK = TRUE
	OK														:	BOOL; //On/Off Delay Signal
	OK_2													:	BOOL; //On/Off Delay Signal 2 - between OK and MonDelOut delay time
	RT														:	BOOL; //R trig based on OK
	FT														:	BOOL; //F trig based on MonDelOut
                            								
//Hardwaresignal       								
	ReadyToRestart											:	BOOL := FALSE; //TRUE when restart of safety circuit is executable 
	MonOut													:	BOOL := FALSE; //output
	MonDelOut												:	BOOL := FALSE; //output delayed
END_STRUCT
END_TYPE

// POUs/Statemodel/eMODE
{attribute 'qualified_only'}
//Default mode enum 0 - 10
{attribute 'to_string'}
TYPE eMODE :
(
	IDLE		 		:= 0,	
	MANUAL				:= 1,
	AUTO				:= 2,
	SEMI_AUTO			:= 3,
	SETUP				:= 4,
	STEP				:= 5,
	PRODUCTION			:= 6,
	MAINTENANCE			:= 7,
	SERVICE				:= 8,
	INIT				:= 9
				
);
END_TYPE

// POUs/Statemodel/eSTATE
{attribute 'qualified_only'}
//Statemodel enum states 0 and 301-320
{attribute 'to_string'}
TYPE eSTATE :
(
	IDLE			:= 0,

	STARTUP			:= 301,
	ABORTING		:= 302,	
	ABORTED			:= 303,
	CLEARING		:= 304,

	STOPPING		:= 305,
	STOPPED			:= 306,
	RESETTING		:= 307,

	STARTING		:= 308,
	STARTED			:= 309,
	EXECUTE			:= 310,
	COMPLETING		:= 311,
	COMPLETE		:= 312,
	
	SUSPENDING		:= 313,
	SUSPENDED		:= 314,
	UNSUSPENDING	:= 315,
	HOLDING			:= 316,
	HELD			:= 317,
	UNHOLDING		:= 318
	);
END_TYPE

// POUs/StringHelper/ExtendedString/T_EXT_STRING
TYPE T_EXT_STRING : STRING(PARAM.MAX_EXT_STRING_LENGTH); END_TYPE

// POUs/StringHelper/ExtendedString/T_EXT_WSTRING
TYPE T_EXT_WSTRING : WSTRING(Param.MAX_EXT_STRING_LENGTH); END_TYPE

// POUs/StringHelper/U_MAX_STRING
TYPE U_MAX_STRING :
UNION
	text				:	STRING(MAX_STRING_LENGTH);
	{attribute 'displaymode':='hex'}
	_BYTES				:	ARRAY[0..MAX_STRING_LENGTH] OF BYTE;	
END_UNION
END_TYPE

// POUs/StringHelper/U_MAX_WSTRING
TYPE U_MAX_WSTRING :
UNION
	text				:	WSTRING(MAX_STRING_LENGTH);
	{attribute 'displaymode':='hex'}
	_BYTES				:	ARRAY[0..MAX_STRING_LENGTH] OF WORD;	
END_UNION
END_TYPE

// GVLs/Gvl
VAR_GLOBAL
	{info <'Please check the disclaimer note vis function DisclaimerStatement (FUN) '>}
	
	CheckBoundsInfo												: 	CheckBoundsInfo; //Checkbounds result buffer 
	EventHandlingStatistic										:	EventHandlingStatisticInfo; //System information of eventlogger 
//	SOURCE_ID													:	SOURCE_ID; //Systemsource ids

	ALWAYS_TRUE										AT  %Q* 	:	BOOL := TRUE;
END_VAR
VAR_GLOBAL CONSTANT
	IBN															: 	BOOL := TRUE;	
END_VAR

// GVLs/PARAM
{attribute 'qualified_only'}
VAR_GLOBAL CONSTANT
//Debug messages											
	ENABLE_DEBUG_MSG_DYNAMIC_MEM_ALLOCATION					:	BOOL := TRUE; //FBs who are allocating memory from the router memory pool via __NEW are writing a message into the ADS logger	

//Controller Tools
	SLIDING_AVERAGE_MAX_ENTRYS								:	INT := 1000;

//String helper
	MAX_EXT_STRING_LENGTH									:	UDINT := 1024; //Max string lenght for extended string FBs (ExtString,ExtWSTRING)	
	XWORD_TO_XXXSTR_EXT_SEPARATOR							:	STRING := '_';

//Data buffer settings
	RINGBUFFER_BYTE_SIMPLE_MAX_BUFFER						:	UINT := 1024;	//Max index byte ringbuffer array
	RINGBUFFER_CHAR_SIMPLE_MAX_BUFFER						:	UINT := 1024;	//Max index byte ringbuffer array for chars 	
	RINGBUFFER_LREAL_SIMPLE_MAX_BUFFER						:	UINT := 10;		//Max index lreal ringbuffer array
	
	FIFO_LREAL_SIMPEL_MAX_BUFFER							:	INT := 10;		//Max index lreal fifo array
	
//File handling 
	READ_DIR_SIMPLE_MAX_ENTRYS								:	INT(1..1000) := 50;	//Max list size of founded files in directory
	READ_DIR_SIMPLE_MAX_STRING_LEN							:	INT := 50;		//Maximum string lenght of files founded in directory
	
//Eventlogger  
	EVENT_HANDLING_CONFIG									:	EVENT_HANDLING_CONFIG  := (
																	GRP_CUSTOMISED_MAX_EVENT			:= 30,		
																	
																	EVENTLOG_READ_MSG_LEN_MIN			:= 0,
																	EVENTLOG_READ_MSG_LEN_MAX			:= 1024,
																	                                    
																	EVENTLOG_READ_MAX_EVENTS			:= 30,		
																	
																	ENABLE_DYNAMIC_EVENT_MSG_FORMAT		:= FALSE,
																	                                    
																	CLASS_NONE_QUIT_REQUIRED			:= FALSE,  	//Class id 0
																	CLASS_MAINTENANCE_QUIT_REQUIRED		:= TRUE,	//Class id 1	
																	CLASS_MESSAGE_QUIT_REQUIRED			:= FALSE,	//Class id 2
																	CLASS_HINT_QUIT_REQUIRED			:= FALSE,	//Class id 3
																	CLASS_STATEINFO_QUIT_REQUIRED		:= FALSE,	//Class id 4
																	CLASS_INSTRUCTION_QUIT_REQUIRED		:= FALSE,	//Class id 5
																	CLASS_WARNING_QUIT_REQUIRED			:= TRUE,	//Class id 6
																	CLASS_ALARM_QUIT_REQUIRED			:= TRUE,	//Class id 7
																	CLASS_PARAMERROR_QUIT_REQUIRED		:= TRUE,	//Class id 8
																	                                    
																	CLASS_NONE_PRIORITY					:= 3,
																	CLASS_MAINTENANCE_PRIORITY			:= 2,
																	CLASS_MESSAGE_PRIORITY				:= 3,
																	CLASS_HINT_PRIORITY					:= 3,
																	CLASS_STATEINFO_PRIORITY			:= 3,
																	CLASS_INSTRUCTION_PRIORITY			:= 3,
																	CLASS_WARNING_PRIORITY				:= 2,   
																	CLASS_ALARM_PRIORITY				:= 1,		
																	CLASS_PARAMERROR_PRIORITY			:= 1);	
		
//Logbook settings 
	LOGBOOK_MAX_DATA										:	INT(1..1000) := 50; //no of messages stored in the PLC - logbook
	LOGBOOK_MAX_MSG_STRING_LENGHT							:	UDINT := 255; //Max sring lenght of logbook message
	LOGBOOK_PUPLISHER_MAX_SUB								:	INT := 5;
	LOGBOOK_SUB_WRT_FILE_LINE_END_SIGN						:	STRING(6) := '$n'; //line end sign
	LOGBOOK_SUB_WRT_FILE_DELAY_FILE_CLOSE					:	TIME := T#5S; //Delay close logbook file and release handle 
	LOGBOOK_SUB_MAX_EVENT_HANDLING							:	UINT(1..100) := 10; //no of EventHandling instances to display logbook entrys
	LOGBOOK_SUB_SEND_MAIL_STR_LINE_END_SIGN					:	STRING(6) := '$r$n'; //line end sign
	
			
//Statemodel control settings
	STATEMODEL_CTRL_MAX_SLAVE								:	INT(1..100) := 8; //no of possible subs for each state model master instance
	
//IO-Fieldbus Master
	ETHERCAT_MASTER_DEV_IO_MAX_FRAMES						:	INT := 4;
	ETHERCAT_DIAG_MAX_SLAVES								:	UINT := 100;
	
	PROFIBUS_MASTER_DEV_IO_MAX_SLAVES						:	INT := 10;
	PROFINET_MASTER_DEV_IO_MAX_BOX							:	INT := 10;

//IO
	ETHERCAT_SLAVE_DEV_FW_UPDATER_MAX_DEV					:	INT := 10;	
	
//Safety 
	SAFETY_PLC_TERM_DIAG_MAX_FB								:	INT := 30;
	SAFETY_IO_TERM_DIAG_MAX									:	INT := 10;
	
//Quicksort settings
	QUICKSORT_MAX_STRING_LENGTH								:	INT := 256;
	QUICKSORT_MAX_WSTRING_LENGTH							:	INT := 256;
	
//Modbus 
	MODBUS_MAX_SLAVE_JOB									:	INT := 10;
	MODBUS_MAX_SLAVES_OF_MASTER								:	INT := 10;
END_VAR

// Version/Global_Version
{attribute 'TcGenerated'}
{attribute 'no-analysis'}
{attribute 'linkalways'}
// This function has been automatically generated from the project information.
VAR_GLOBAL CONSTANT
	{attribute 'const_non_replaced'}
	stLibVersion_EngineeringToolbox : ST_LibVersion := (iMajor := 3, iMinor := 1, iBuild := 0, iRevision := 4, nFlags := 0, sVersion := '3.1.0.4');
END_VAR

// POUs/_Miscellaneous/64BitFunctions/CLEARBIT64
{attribute 'displaymode':='binary'}	
FUNCTION CLEARBIT64 : LWORD
VAR_INPUT
	inVal64			:	LWORD;
	bitNo			:	INT;
END_VAR
VAR
{attribute 'displaymode':='binary'}	
	lwConst 			:	LWORD := 1;
END_VAR

CLEARBIT64 := inVal64 AND NOT (SHL(lwConst,bitNo MOD 64));

END_FUNCTION

// POUs/_Miscellaneous/64BitFunctions/CSETBIT64
{attribute 'displaymode':='binary'}	
FUNCTION CSETBIT64 : LWORD (* conditional set bit in 64bit lword *)
VAR_INPUT
	inVal64													:	LWORD;
	bitNo													:	INT;
	bitVal													:	BOOL;		(* value to which the bit should be set *)
END_VAR
VAR
{attribute 'displaymode':='binary'}	
	lwConst 												: 	LWORD := 1;
END_VAR

IF bitVal
THEN
	CSETBIT64 												:= inVal64 OR SHL(lwConst,bitNo MOD 64);
ELSE
	CSETBIT64 												:= inVal64 AND NOT (SHL(lwConst,bitNo MOD 64));
END_IF;

END_FUNCTION

// POUs/_Miscellaneous/64BitFunctions/GETBIT64
{attribute 'displaymode':='binary'}	
FUNCTION GETBIT64 : BOOL
VAR_INPUT
	inVal64												:	LWORD;
	bitNo												:	INT;
END_VAR
VAR
{attribute 'displaymode':='binary'}	
	lwConst			 									: 	LWORD := 1;
END_VAR

GETBIT64												:= ( inVal64 AND SHL(  lwConst,bitNo MOD 64 ) ) > 0;

END_FUNCTION

// POUs/_Miscellaneous/64BitFunctions/SETBIT64
{attribute 'displaymode':='binary'}	
FUNCTION SETBIT64 : LWORD
VAR_INPUT
	inVal64													:	LWORD;
	bitNo													:	INT;
END_VAR
VAR
{attribute 'displaymode':='binary'}	
	lwConst 												: 	LWORD := 1;
END_VAR

SETBIT64 															:= inVal64 OR SHL( lwConst,bitNo MOD 64 );

END_FUNCTION

// POUs/_Miscellaneous/Conversions/ADSERROR_TO_WIN32ERROR
{attribute 'no_check'}
//Read win 32 errorcode incl. win socket error from ADS error code (IDs >= 16#8007000)
FUNCTION ADSERROR_TO_WIN32ERROR : UDINT
VAR_INPUT
{attribute 'displaymode':='hex'}
	ErrorID													:	UDINT;
END_VAR
VAR
END_VAR

IF ErrorID >= TO_UDINT(16#80070000) AND ErrorID <= TO_UDINT(16#8007FFFF)
THEN	
	ADSERROR_TO_WIN32ERROR									:= ErrorID - TO_UDINT(16#80070000);
ELSE
	ADSERROR_TO_WIN32ERROR									:= ErrorID;
END_IF

END_FUNCTION

// POUs/_Miscellaneous/WIN
{attribute 'monitoring' := 'variable'}
{attribute 'no_check'}
//if X between LO and HI then win = True else win = false
FUNCTION WIN : BOOL
VAR_INPUT
	X		: LREAL ;	
	LO		: LREAL ;
	HI		: LREAL ;
END_VAR
VAR
END_VAR

	(* window check 			  											ds	*)
	(****************************************************************************)
	(* if X between LO and HI then win = True else win = false					*)
	(****************************************************************************)


(* the current value of the window  *****************************************)
WIN 														:= 		X >= LO AND X <= HI;
(*****************************************************************************)

END_FUNCTION

// POUs/_Miscellaneous/Conversions/ADSERROR_TO_WSERROR
{attribute 'no_check'}
//Convert ADS error id into winsocket error enum
FUNCTION ADSERROR_TO_WSERROR : E_WinsockError
VAR_INPUT
{attribute 'displaymode':='hex'}
	ErrorID													: UDINT;
END_VAR
VAR
END_VAR

IF ErrorID >= TO_UDINT(16#80070000) AND ErrorID <= TO_UDINT(16#8007FFFF)
THEN
	ADSERROR_TO_WSERROR										:= TO_INT(ErrorID - TO_UDINT(16#80070000));
	IF ADSERROR_TO_WSERROR < 10004 OR ADSERROR_TO_WSERROR >= 12000
	THEN //Because of other Win32 error
		ADSERROR_TO_WSERROR									:= WSOK;
	END_IF
ELSIF ErrorID = 16#274C
THEN
	ADSERROR_TO_WSERROR										:= WSAETIMEDOUT;
ELSIF ErrorID = 16#274D
THEN
	ADSERROR_TO_WSERROR										:= WSAECONNREFUSED;
ELSIF ErrorID = 16#2751
THEN
	ADSERROR_TO_WSERROR										:= WSAEHOSTUNREACH;
ELSIF ErrorID >= TO_UDINT(16#00008000) AND ErrorID <= TO_UDINT(16#000080FF)
THEN //Internal error TCP/IP Server 
	ADSERROR_TO_WSERROR										:= WSAEHOSTUNREACH;
ELSE
	ADSERROR_TO_WSERROR										:= WSOK;
END_IF

END_FUNCTION

// POUs/_Miscellaneous/Conversions/C_TO_F
//Converts Celsius into Fahrenheit
FUNCTION C_TO_F : LREAL
VAR_INPUT
	C														:	LREAL; //Celsius
END_VAR
VAR
END_VAR

C_TO_F := C * 1.8 + 32.0;

END_FUNCTION

// POUs/_Miscellaneous/Conversions/DEGREES_TO_RPM
{attribute 'no_check'}
//°/s -> RPM
FUNCTION DEGREES_TO_RPM : LREAL
VAR_INPUT
	IN														:	LREAL;	//Input value
END_VAR
VAR
END_VAR

DEGREES_TO_RPM 											:= IN * 60.0 / 360.0;

END_FUNCTION

// POUs/IO/Input
{attribute 'no_check'}
FUNCTION_BLOCK Input
VAR_INPUT
	Force													:	BOOL := FALSE; 	//simulates Input
	Invert													:	BOOL := FALSE; 	//inverts the Hardware Input
	PT_ON													:	TIME := T#0MS;	//on delay
	PT_OFF													:	TIME := T#0MS;	//off delay
END_VAR             										
VAR_OUTPUT          										
	Q														:	BOOL;	//Signal Delay
	Q_RT													:	BOOL;	//R_Trig Signal of Q
	Q_FT													:	BOOL;	//F_Trig Signal of Q
	Q_DIRECT												:	BOOL; 	//Signal direct
	In												AT  %I* : 	BOOL; 	//Hardware Input
END_VAR
VAR
	TON														:	TON;
END_VAR

(* Input/Sensor Functionblock with On/Off	attenuation and rising / fallen edge 	V2.0	*)
(********************************************************************************************)

(************************************)
IF NOT Q THEN
	TON(IN := (IN OR Force) XOR Invert, PT := PT_ON);
	Q 														:= TON.Q;
	Q_RT 													:= Q;
	Q_FT 													:= FALSE;
	Q_DIRECT 												:= TON.IN;
ELSE
	TON(IN := NOT ((IN OR Force) XOR Invert), PT := PT_OFF);
	Q 														:= Q AND NOT TON.Q;
	Q_RT 													:= FALSE;
	Q_FT 													:= NOT Q;
	Q_DIRECT 												:= Q AND NOT TON.IN;
END_IF
(********************************************************************************************)

END_FUNCTION_BLOCK

// POUs/_Miscellaneous/Conversions/DWORD_TO_REAL_EX
// Converts a 32bit float variable with swapped words into a TwinCAT conform REAL value after checking whether the result will be a valid number
// Use PDWORD_TO_DWORD in case the source variable is e..g a byte array -> RealVar := DWORD_TO_REAL_EX(In := PDWORD_TO_DWORD(ADR(ModBusCom.Data[1]));
FUNCTION DWORD_TO_REAL_EX : REAL
VAR_INPUT
	In						:	DWORD;
END_VAR
VAR
	Dummy					: U_32BIT_DATATYPE;
END_VAR


	Dummy._DWORD			:= In;

	F_SwapRealEx(Dummy._REAL);

	IF	IsFinite(F_REAL(Dummy._REAL)) THEN
		DWORD_TO_REAL_EX := Dummy._REAL;
	ELSE
		DWORD_TO_REAL_EX := 0.0;
	END_IF

END_FUNCTION

// POUs/_Miscellaneous/Conversions/F_TO_C
//Convert Fahrenheit into Celsius
FUNCTION F_TO_C : LREAL
VAR_INPUT
	F														:	LREAL; //Fahrenheit
END_VAR
VAR
END_VAR

F_TO_C := (F - 32.0) * 0.5555555555555;

END_FUNCTION

// POUs/_Miscellaneous/Conversions/GF_TO_N
{attribute 'no_check'}
//Gram-force to newton
FUNCTION GF_TO_N : LREAL
VAR_INPUT
	GF				:	LREAL;
END_VAR
VAR
END_VAR
(*
Gram-force to newton (gf to N):
Fn = Fgf ×0.00980665
Example:
If gf = 156 then N = 1.5298374N

Newton to gram-force (N to gf):
Fgf = Fn / 0.00980665
*)

GF_TO_N := GF * 0.00980664999999998 ;

END_FUNCTION

// POUs/_Miscellaneous/Conversions/HRESULT_TO_ADSERROR
FUNCTION HRESULT_TO_ADSERROR     : E_AdsErr //Returns ADS error code from HRESULT (HRESULT HighWord offset = 16#9811, values <0 = Error, ==0 = OK, >0 = OK with Info   
VAR_INPUT
{attribute 'displaymode':='hex'}
	hr									:	HRESULT;
END_VAR
VAR
END_VAR

IF hr >= TO_DINT(16#98110000)
	AND hr <= TO_DINT(16#9811FFFF) 
THEN	
	HRESULT_TO_ADSERROR				:= TO_UDINT(hr - TO_DINT(16#98110000));
ELSE
	HRESULT_TO_ADSERROR				:= E_AdsErr.NOERR; //No ADS Error
END_IF

END_FUNCTION

// POUs/_Miscellaneous/Conversions/LWORD_TO_LREAL_EX
// Converts a 64bit double variable with swapped words into a TwinCAT conform LREAL value after checking whether the result will be a valid number
// Use PLWORD_TO_LWORD in case the source variable is e..g a byte array -> LRealVar := LWORD_TO_LREAL_EX(In := PLWORD_TO_LWORD(ADR(ModBusCom.Data[1]));
FUNCTION LWORD_TO_LREAL_EX : LREAL
VAR_INPUT
	In						: LWORD;
END_VAR
VAR
	Dummy					: U_64BIT_DATATYPE;
END_VAR

	Dummy._LWORD			:= In;
	Dummy._LWORD			:= SWAP_WORDS_OF_LWORD(Dummy._LWORD);
	
	IF	IsFinite(F_LREAL(dummy._LREAL)) THEN
		LWORD_TO_LREAL_EX 	:= dummy._LREAL;
	ELSE
		LWORD_TO_LREAL_EX	:= 0.0;
	END_IF

END_FUNCTION

// POUs/_Miscellaneous/Conversions/SWAP_WORDS_OF_LWORD
// Returns TRUE when words are successfully swapped 
FUNCTION SWAP_WORDS_OF_LWORD : LWORD
VAR_INPUT
	in														:	LWORD;
END_VAR
VAR
	pTmp													:	POINTER TO WORD;
	WordArray												:	ARRAY[1..4] OF WORD;
END_VAR

	pTmp													:= ADR(in);
	WordArray[4]											:= pTmp^; // [1]
	pTmp													:= pTmp + 2;
	WordArray[3]											:= pTmp^; // [2]
	pTmp													:= pTmp + 2;
	WordArray[2]											:= pTmp^; // [3]
	pTmp													:= pTmp + 2;
	WordArray[1]											:= pTmp^; // [4]
	
	Memcpy(ADR(SWAP_WORDS_OF_LWORD),ADR(WordArray),SIZEOF(WordArray));

END_FUNCTION

// POUs/_Miscellaneous/Conversions/MMIN_TO_MMS
{attribute 'no_check'}
//m/min -> mm/s
FUNCTION MMIN_TO_MMS : LREAL
VAR_INPUT
	IN														:	LREAL;	//Input value
END_VAR
VAR
END_VAR

MMIN_TO_MMS 												:= IN * 1000.0 / 60.0;

END_FUNCTION

// POUs/_Miscellaneous/Conversions/MMS_TO_MMIN
{attribute 'no_check'}
//mm/s -> m/min
FUNCTION MMS_TO_MMIN : LREAL
VAR_INPUT
	IN														:	LREAL;	//Input value
END_VAR
VAR
END_VAR

MMS_TO_MMIN 												:= IN * 0.001 * 60;

END_FUNCTION

// POUs/_Miscellaneous/Conversions/N_TO_GF
{attribute 'no_check'}
//Newton to Gram-force
FUNCTION N_TO_GF : LREAL
VAR_INPUT
	FN				:	LREAL;
END_VAR
VAR
END_VAR
(*
Gram-force to newton (gf to N):
Fn = Fgf ×0.00980665
Example:
If gf = 156 then N = 1.5298374N

Newton to gram-force (N to gf):
Fgf = Fn / 0.00980665
*)

N_TO_GF := FN / 0.00980664999999998;

END_FUNCTION

// POUs/_Miscellaneous/Conversions/REAL_TO_FMLREAL
{attribute 'no_check'}
//Limit the number of decimal places in a lreal variable   
FUNCTION REAL_TO_FMLREAL : LREAL
VAR_INPUT
	 In														:	REAL;	//Input value
	 Digits													:	INT;	//number of digits to be shown
END_VAR     												
VAR         												
	 Faktor													:	LREAL;
END_VAR

Faktor														:=	EXPT(10,ABS(Digits));
IF Faktor = 0.0
THEN
	REAL_TO_FMLREAL 										:= 0.0;
ELSE
	REAL_TO_FMLREAL 										:= LINT_TO_LREAL(LREAL_TO_LINT(IN * Faktor)) / Faktor;
END_IF

END_FUNCTION

// POUs/_Miscellaneous/Conversions/RPM_TO_DEGREES
{attribute 'no_check'}
//RPM -> °/s
FUNCTION RPM_TO_DEGREES : LREAL
VAR_INPUT
	IN														:	LREAL;	//Input value
END_VAR
VAR
END_VAR

RPM_TO_DEGREES 												:= IN * 360.0 / 60.0	;

END_FUNCTION

// POUs/_Miscellaneous/Conversions/SWAP_BYTES_OF_WORDS
//Swapping bytes in an array of words  
FUNCTION SWAP_BYTES_OF_WORDS : BOOL
VAR_INPUT
	pIn														:	POINTER TO WORD;
	NoOfWords												:	INT;
END_VAR
VAR
	pTemp													:	POINTER TO WORD;
	i														:	INT; 
END_VAR

IF pIn <> 0 THEN
	FOR i := 1 TO NoOfWords BY 2 DO 
		pTemp													:= pIn + TO_WORD(i-1);
		pTemp^ 													:= HOST_TO_BE16(pTemp^);	
	END_FOR
	SWAP_BYTES_OF_WORDS											:= TRUE;
ELSE
	SWAP_BYTES_OF_WORDS											:= FALSE;
END_IF

END_FUNCTION

// POUs/_Miscellaneous/Conversions/SWAP_WORDS_OF_DWORD
//Swaps high and low word of an DWORD variable
FUNCTION SWAP_WORDS_OF_DWORD : DWORD
VAR_INPUT
	in														:	DWORD;
END_VAR
VAR
	pTmp													:	POINTER TO WORD;
	WordArray												:	ARRAY[1..2] OF WORD;
	i														:	INT; 
END_VAR

	ptmp														:= ADR(In);
	WordArray[2]												:= ptmp^; // [1]
	ptmp														:= ptmp + 2;
	WordArray[1]												:= ptmp^; // [2]

	MEMCPY(ADR(SWAP_WORDS_OF_DWORD),ADR(WordArray),SIZEOF(WordArray));

END_FUNCTION

// POUs/_Miscellaneous/Conversions/TO_FMLREAL
{attribute 'no_check'}
//Limits the number of decimal places in a floating point variable 
//or converts an integer number into a LREAL variable with with corresponding decimal places 
FUNCTION TO_FMLREAL : LREAL
VAR_INPUT
	 In														:	ANY_NUM;	//Input value
	 Digits													:	INT (1..32);	//number of digits to be shown
END_VAR     												
VAR         												
	 Factor													:	LREAL;
	 Value													:	LREAL;
END_VAR



IF Digits <= 0
THEN
	TO_FMLREAL												:= 0.0;	
ELSIF In.TypeClass = __SYSTEM.TYPE_CLASS.TYPE_LREAL
THEN
	Factor													:=EXPT(10,Digits);
	TO_FMLREAL												:= LINT_TO_LREAL(LREAL_TO_LINT(PLREAL_TO_LREAL(IN.pValue) * Factor)) / Factor;
ELSIF In.TypeClass = __SYSTEM.TYPE_CLASS.TYPE_REAL
THEN
	Factor													:=EXPT(10,Digits);
	TO_FMLREAL												:= LINT_TO_LREAL(LREAL_TO_LINT(PREAL_TO_REAL(IN.pValue) * Factor)) / Factor;
ELSE // Integer
	Factor													:=EXPT(10,Digits);
	CASE in.TypeClass OF		
	__SYSTEM.TYPE_CLASS.TYPE_USINT:	Value					:= TO_LREAL(PUSINT_TO_USINT(IN.pValue));								
	__SYSTEM.TYPE_CLASS.TYPE_UINT:	Value					:= TO_LREAL(PUINT_TO_UINT(IN.pValue));	
	__SYSTEM.TYPE_CLASS.TYPE_UDINT:	Value					:= TO_LREAL(PUDINT_TO_UDINT(IN.pValue));	
	__SYSTEM.TYPE_CLASS.TYPE_ULINT:	Value					:= TO_LREAL(PULINT_TO_ULINT(IN.pValue));	
	__SYSTEM.TYPE_CLASS.TYPE_SINT:	Value					:= TO_LREAL(PSINT_TO_SINT(IN.pValue));	
	__SYSTEM.TYPE_CLASS.TYPE_INT:	Value					:= TO_LREAL(PINT_TO_INT(IN.pValue));	
	__SYSTEM.TYPE_CLASS.TYPE_DINT:	Value					:= TO_LREAL(PDINT_TO_DINT(IN.pValue));	
	__SYSTEM.TYPE_CLASS.TYPE_LINT:	Value					:= TO_LREAL(PLINT_TO_LINT(IN.pValue));	
	ELSE
		TO_FMLREAL											:= 0.0;
		RETURN;
	END_CASE

	TO_FMLREAL												:= Value / Factor;
END_IF

END_FUNCTION

// POUs/_Miscellaneous/CAM
{attribute 'monitoring' := 'variable'}
{attribute 'no_check'}
//if x in setpoint +/- window then cam = true else cam = false
FUNCTION CAM : BOOL
VAR_INPUT
	X														: LREAL ; 	//value to be monitored
	SETP													: LREAL ;	//target value
	WINDOW													: LREAL ;	//tolerance zone
END_VAR
VAR
END_VAR

(* cam check				  											ds	*)
(****************************************************************************)
(* if x in setpoint +/- window then cam = true else cam = false				*)
(****************************************************************************)

(* the current value of the window  *****************************************)
CAM 														:=  X >= SETP - WINDOW AND X <= SETP + WINDOW ;
(****************************************************************************)

END_FUNCTION

// POUs/_Miscellaneous/CAM3D
{attribute 'monitoring' := 'variable'}
{attribute 'no_check'}
//if x,y,z in setpoint +/- window then cam3d = true else cam3d = false	
FUNCTION CAM3D : BOOL
VAR_INPUT
	X														: LREAL ;	//X-value to be monitored
	Y														: LREAL;	//Y-value to be monitored
	Z														: LREAL;	//Z-value to be monitored
	SETP_X													: LREAL ;	//X-target value
	SETP_Y													: LREAL ;	//Y-target value
	SETP_Z													: LREAL ;	//Z-target value
	WINDOW													: LREAL ;	//tolerance zone
END_VAR
VAR
END_VAR

	(* cam check				  											ds	*)
	(****************************************************************************)
	(* if x in setpoint +/- window then cam = true else cam = false				*)
	(****************************************************************************)

(* the current value of the window  *****************************************)
CAM3D 														:=  	X >= SETP_X - WINDOW AND X <= SETP_X + WINDOW
																AND Y >= SETP_Y - WINDOW AND Y <= SETP_Y + WINDOW
																AND Z >= SETP_Z - WINDOW AND Z <= SETP_Z + WINDOW;

(******************************************************************************)

END_FUNCTION

// POUs/_Miscellaneous/ERROR_HDL
{attribute 'no_check'}
//Error handle object to collect/provide additional error information like state , function name, id or information text 
FUNCTION_BLOCK ERROR_HDL
VAR_INPUT
	Flag													:	BOOL := FALSE; 	//Error is active
	SourceId												: 	UDINT := 0; 	//Source ID for EventLogger if neede
	Class													:	E_TcEventClass := TC2_SYSTEM.TCEVENTCLASS_ALARM;
{attribute 'displaymode':='hex'}
	Id														:	DINT := 0;	//Error id 
	State													:	DINT := 0;	//State where error occures
	Text													:	STRING(MAX_STRING_LENGTH) :='';	//Information text
	Fnc														:	STRING(20) :='';	//Function name of error source
END_VAR
VAR_OUTPUT
END_VAR
VAR
END_VAR

;

//Reset all entrys to zero/empty
METHOD PUBLIC reset : BOOL  //Return value = TRUE if execution finished
VAR_INPUT
END_VAR
flag 														:= FALSE;
SourceId													:=0;
class 														:= TC2_SYSTEM.TCEVENTCLASS_NONE;
id															:=0;
state														:=0;
text														:='';
fnc															:='';
Reset														:= TRUE;
END_METHOD

END_FUNCTION_BLOCK

// POUs/_Miscellaneous/FbBase
//Template for PlcOpen FB implementations - Extend final implementations from this FB
FUNCTION_BLOCK FbBase EXTENDS FbBaseOutputs
VAR_INPUT
	Execute													:	BOOL := FALSE; //The function block starts execution with a rising edge on this input  
END_VAR
VAR_IN_OUT
END_VAR
VAR_OUTPUT
END_VAR
VAR 
END_VAR
VAR
(* Cache ********************************************************************************)
	State													: INT := 0;

(* Trigger ******************************************************************************)
	rtExecute												:	R_TRIG;	

(* Dummys *******************************************************************************)

END_VAR

END_FUNCTION_BLOCK

// POUs/_Miscellaneous/FbBaseOutputs
//Template for PlcOpen FB implementations - Extend final implementations from this FB
FUNCTION_BLOCK FbBaseOutputs
VAR_INPUT
END_VAR
VAR_IN_OUT
END_VAR
VAR_OUTPUT
	Busy													: BOOL; // Busy is TRUE at the rising edge of Execute and stays TRUE as long as the FB is performing any action and must be called cyclically to be executed.
	Done													: BOOL; // Is TRUE if FB was executed successfully and stays TRIE for min one cylce or as long as Execute is set to true  
	Error													: BOOL;	// Is TRUE when an error occurred during the execution of the Function Block 
{attribute 'displaymode':='hex'}  
	ErrorId													: UDINT; //Error identification - see e.g. ADS return codes at Beckhoff infosys for further information 
END_VAR
VAR 
END_VAR
VAR
END_VAR

END_FUNCTION_BLOCK

// POUs/_Miscellaneous/FbBaseExt
//Template for PlcOpen FB implementations with local path variable filled by attribute 'instance-path'
{attribute 'reflection'}
FUNCTION_BLOCK FbBaseExt EXTENDS FbBase
VAR_INPUT
END_VAR
VAR_IN_OUT
END_VAR
VAR_OUTPUT
    {attribute 'instance-path'}
    {attribute 'no_init'}
    Path  													: STRING;
END_VAR
VAR 
END_VAR
VAR
END_VAR

END_FUNCTION_BLOCK

// POUs/_Miscellaneous/getNoOfBits
//Returns number of bits set in integer data type variable 
FUNCTION getNoOfBits : INT 
VAR_INPUT
	In														:	ANY_INT;
END_VAR
VAR
{attribute 'displaymode':='binary'}		
	_ULINT													: 	ULINT;	
END_VAR

	getNoOfBits												:= 0;
	MEMCPY(ADR(_ULINT) + (SIZEOF(_ULINT) - TO_UDINT(IN.diSize)),In.pValue,TO_UDINT(IN.diSize));
	WHILE (_ULINT > 0) DO
		_ULINT 												:= _ULINT AND (_ULINT -1); 
		getNoOfBits											:= getNoOfBits + 1;
	END_WHILE

END_FUNCTION

// POUs/_Miscellaneous/LOGx
//The function returns the base 2 logarithm of a number 
//Permitted data types for the input variables: any numeric basic data type
FUNCTION LOGx : LREAL
VAR_INPUT
	In														: LREAL;
	Basis													: UINT;
END_VAR
VAR
END_VAR

IF Basis = 0 OR In <= 0.0
THEN
	LOGx													:= 0.0;
ELSE
	LOGx 													:= LOG(In) / LOG(Basis);
END_IF

END_FUNCTION

// POUs/_Miscellaneous/OEECalculation
//Overall Equipment Effectiveness - see www.OEE.com
//The preferred OEE calculation is based on the three OEE Factors: Availability, Performance, and Quality
//It takes into account all losses, resulting in a measure of truly productive manufacturing time. It is calculated as
//
//Availability:
//Takes into account all events that stop planned production long enough where it makes sense to track a reason for being down (typically several minutes).
//
//Performance:
//Takes into account anything that causes the manufacturing process to run at less than the maximum possible speed when it is running (including both Slow Cycles and Small Stops).
//
//Quality:
//Takes into account manufactured parts that do not meet quality standards, including parts that need rework. 
//
{attribute 'no_check'}
FUNCTION_BLOCK OEECalculation
VAR_INPUT
	ResetCalc												:	BOOL; //Reset all values
	PlannedProdTime											:	TIME; //Total time that equipment is expected to produce. Calculated by subtracting Schedule Loss from All time Benchmark that OEE is measured against
	IdealCycleTime											:	TIME; //Theoretical minimum time to produce ONE unit (Reciprocal of Ideal run rate).	
	ProdRunning												:	BOOL; //TRUE to record elapsed actual production time / Do not use if actual production time will be set by attribute "ActualProdTime"	
	ProdPausing												:	BOOL; //TRUE to record allowed machine stop which will be not tracked as down time (Caused by unexpected stops)	
END_VAR
VAR_OUTPUT
	TotalUnitCount											:	LREAL; 
	GoodUnitCount											:	LREAL; 
	BadUnitCount											:	LREAL; 
	DownTime												:	TIME;  //= PlannedProdTime - ActualProdTime - ActualPauseTime. All time where the manufactoring process was intended to be running but was not due to unplanned stops (Stop time)
	Availability											:	LREAL; //= Ratio of ActualProdTime / PlannedProdTime in %
	Performance												:	LREAL; //= Ratio of (IdealCycleTime x TotalUnitCount) / ActualProdTime in %
	Quality													:	LREAL; //= Ratio of GoodUnitCount / TotalUnitCount in %
	Summary													:	LREAL; //= Result of (Availability x Performance x Quality( or ((GoodUnitCount x IdealCycleTime) / PlannedProdTime) in %
	InProduction											:	BOOL; //Accumulating actual production time 
	InPausing												:	BOOL; //Pausing time running, elapsed time will not be a part of stop time (Down time)
	Error													:	BOOL; //Invalid parameter e.g. Any value > 100% , Actual prod. time > Planned prod. time, Bad unit count > total unit count
END_VAR
VAR
	ProdTime												:	TIME; //The manufactoring process is scheduled for production and is running. Calculated by subtracting down time.
	PauseTime												:	TIME;
	IdealRunRate											:	LREAL; //Theoretical maximum prodcution rate (Reciprocal of Ideal cylce time)
	AvailabilityRate										:	LREAL; 
	PerformanceRate											:	LREAL; 
	QualityRate												:	LREAL; 
	SummaryRate												:	LREAL;
	ActSysTime												:	TIME;
	LastSysTime												:	TIME;	
	rfProdRunning											:	RF_TRIG;
	rfPauseRunning											:	RF_TRIG;
END_VAR

	(* Calculate overall equipment effectivness 				*)
	(************************************************************)

(* Reset *****************************************************************)
	IF ResetCalc THEN reset(); END_IF
	
(* Get intern values *******************************************************)
	IdealRunRate											:= SEL(IdealCycleTime = T#0MS,  1.0 / TO_LREAL(IdealCycleTime), 0.0);
	BadUnitCount											:= TotalUnitCount - GoodUnitCount ;

(* Record production time, pausing and resulting down time *******************)
	rfProdRunning(CLK := ProdRunning); rfPauseRunning(CLK := ProdPausing);
	IF rfProdRunning.Q 
	THEN
		InProduction										:= ProdRunning ;
		InPausing											:= FALSE;
	ELSIF rfPauseRunning.Q
	THEN
		InProduction										:= FALSE ;
		InPausing											:= ProdPausing;		
	END_IF
	
	ActSysTime 												:= TIME();(* read system time *)
	IF InProduction 
	THEN	
		ProdTime		 									:= (ActSysTime - LastSysTime) + ProdTime;  (* add the current milliseconds *)		
	ELSIF InPausing
	THEN
		PauseTime		 									:= (ActSysTime - LastSysTime) + PauseTime;  (* add the current milliseconds *)		
	END_IF
	LastSysTime 											:= ActSysTime;

	//Final issue caused down time
	DownTime												:= MAX(T#0MS, PlannedProdTime - ProdTime - PauseTime);

(* Calculate availability ********************************************)
	IF PlannedProdTime = T#0MS
	THEN
		AvailabilityRate									:= 0.0;
	ELSE
		AvailabilityRate									:= TO_LREAL(ProdTime) / TO_LREAL(PlannedProdTime);	
	END_IF
	Availability											:= AvailabilityRate * 100.0;
					
(* Calcualate performance ********************************************)					
	IF ProdTime = T#0MS OR IdealRunRate = 0.0
	THEN
		PerformanceRate										:= 0.0;	
	ELSE
		PerformanceRate										:= (TotalUnitCount/TO_LREAL(ProdTime) / IdealRunRate);	
	END_IF
	Performance												:= PerformanceRate * 100.0;
	
(* Calcualte quality *****************************************************)
	IF TotalUnitCount = 0.0
	THEN
		QualityRate											:= 0.0;	
	ELSE
		QualityRate											:= GoodUnitCount / TotalUnitCount;		
	END_IF
	Quality													:= QualityRate * 100.0;
	
(* OEE Result *************************************************************)
	SummaryRate												:= AvailabilityRate * PerformanceRate * QualityRate;
	Summary													:= SummaryRate * 100.0;
	
	Error													:= AvailabilityRate > 1.0 OR PerformanceRate > 1.0 OR QualityRate > 1.0 OR ProdRunning AND ProdPausing OR BadUnitCount < 0.0;

(****************************************************************************)

METHOD PUBLIC addBadUnits : BOOL  //Return value = TRUE if execution finished
VAR_INPUT
	NoOfUnits										:	LREAL;
END_VAR
BadUnitCount										:= BadUnitCount + NoOfUnits;
TotalUnitCount										:= BadUnitCount + GoodUnitCount;
addBadUnits											:= TRUE;
END_METHOD

METHOD PUBLIC addGoodUnits : BOOL //Return value = TRUE if execution finished
VAR_INPUT
	NoOfUnits										:	LREAL;
END_VAR
GoodUnitCount										:= GoodUnitCount + NoOfUnits;
TotalUnitCount										:= BadUnitCount + GoodUnitCount;
addGoodUnits										:= TRUE;
END_METHOD

METHOD PUBLIC reset : BOOL //Return value = TRUE if execution finished
VAR_INPUT
END_VAR

	
	//Reset memory
	ProdTime												:= T#0MS;
	PauseTime												:= T#0MS; 
	TotalUnitCount											:= 0.0;
	BadUnitCount											:= 0.0;
	GoodUnitCount											:= 0.0;
	AvailabilityRate										:= 0.0;
	PerformanceRate											:= 0.0;
	QualityRate												:= 0.0;
	SummaryRate												:= 0.0;
		
	//Reset outputs values
	IdealRunRate											:= 0.0;
	GoodUnitCount											:= 0.0;
	DownTime												:= T#0MS;
	Availability											:= 0.0;
	Performance												:= 0.0;
	Quality													:= 0.0;
	Summary													:= 0.0;
	InPausing												:= FALSE;
	InProduction											:= FALSE;
	Error													:= FALSE;
	
	reset													:= TRUE;
END_METHOD

END_FUNCTION_BLOCK

// POUs/_Miscellaneous/RF_TRIG
{attribute 'no_check'}
//Rising and falling trigger
FUNCTION_BLOCK RF_TRIG
VAR_INPUT
	CLK										:	BOOL;
END_VAR
VAR_OUTPUT
	M										:	BOOL;
	Q										:	BOOL;
END_VAR
VAR
END_VAR

IF CLK XOR M
THEN
	M										:= NOT M;
	Q										:= TRUE;
ELSE
	Q										:= FALSE;	
END_IF

END_FUNCTION_BLOCK

// POUs/_Miscellaneous/polynomial
//calculate polynomial of certain degree
// y := p0 + p1*x^1 + p2*x^2 + p3*x^3 + p4*x^4 + p5*x^5 + p6*x^6 + p7*x^7 + p8*x^8;
FUNCTION polynomial : LREAL 							
VAR_INPUT
	X			: LREAL;
	Degree		: INT;

	p0			: LREAL;
	p1			: LREAL;
	p2			: LREAL;
	p3			: LREAL;
	p4			: LREAL;
	p5			: LREAL;
	p6			: LREAL;
	p7			: LREAL;
	p8			: LREAL;
END_VAR
VAR
END_VAR


IF degree >= 0 THEN Polynomial := 				p0 			  ; 	ELSE RETURN; END_IF
IF degree >= 1 THEN Polynomial := Polynomial + 	p1 * EXPT(x,1); 	ELSE RETURN; END_IF
IF degree >= 2 THEN Polynomial := Polynomial + 	p2 * EXPT(x,2); 	ELSE RETURN; END_IF
IF degree >= 3 THEN Polynomial := Polynomial + 	p3 * EXPT(x,3); 	ELSE RETURN; END_IF
IF degree >= 4 THEN Polynomial := Polynomial + 	p4 * EXPT(x,4); 	ELSE RETURN; END_IF
IF degree >= 5 THEN Polynomial := Polynomial + 	p5 * EXPT(x,5); 	ELSE RETURN; END_IF
IF degree >= 6 THEN Polynomial := Polynomial + 	p6 * EXPT(x,6); 	ELSE RETURN; END_IF
IF degree >= 7 THEN Polynomial := Polynomial + 	p7 * EXPT(x,7); 	ELSE RETURN; END_IF
IF degree >= 8 THEN Polynomial := Polynomial + 	p8 * EXPT(x,8); 	ELSE RETURN; END_IF

END_FUNCTION

// POUs/_Miscellaneous/scale
//Discription:	"SCALE" scales the In-Value, which goes from InLow to InHigh, between the commited OutLow and OutHigh range.
//Used for AnalogIn/Out
FUNCTION scale : LREAL
VAR_INPUT
	In				 										: LREAL;
	InLow 													: LREAL;
	InHigh 													: LREAL;
	OutLow 													: LREAL;
	OutHigh 												: LREAL;
END_VAR
VAR
	Lim														: LREAL;
	X														: LREAL;
END_VAR

IF OutHigh <> OutLow 
THEN
	X														:= InHigh - InLow;
	IF x <> 0.0             									
	THEN       
		Lim 												:= LIMIT(InLow,In,InHigh) - InLow;             									
		X		 											:= (OutHigh - OutLow) / X;
		scale 												:= (X * Lim) + OutLow;			
	ELSE                    									
		scale												:= 0.0;
	END_IF
ELSE
	scale													:= 0.0;	
END_IF

END_FUNCTION

// POUs/IO/AnalogIn
{attribute 'no_check'}
FUNCTION_BLOCK AnalogIn
VAR_INPUT
	MinValue												: 	LREAL 	:= 0.0;
	MaxValue												: 	LREAL 	:= 0.0;
	NoOfDigits												: 	INT 	(0..10)	:= 0; 	//number of decimal digits of scaled Q variable 
	OutOnError												:	LREAL 	:= 0.000000000000000001;
{attribute 'displaymode':='binary'}                     	
	Options													:	BYTE  := 2#0000_0000; 	//.0 = FALSE scalve value from 0 <-> 32767 / TRUE scale value with sign -32768 <-> 32767
	Offset													:	LREAL := 0.0;
END_VAR                 									
VAR                                                     	
{attribute 'displaymode':='binary'}                     	
	Status										AT  %I*		:	WORD := 2#0000_0000_0000_0000; //Terminal status word -> can also be linked with status byte 
END_VAR                                                 	
VAR_OUTPUT                                              	
	Q														:	LREAL;		//Scaled result value
	In											AT  %I* 	: 	INT; 		//Hardware Input

	(* Status bit *)
	Underrange 												:	BOOL;	//Bit 0
	Overrange												:	BOOL;	//Bit 1
	Limit_1													:	BYTE;(* Bit 2-3 			0: not active
																						1: value is smaller than limit 
																						2: value is bigger than limit 
																						3: value is equal to limit  *)
	Limit_2													:	BYTE;(* Bit 4-5 			0: not active
																						1: value is smaller than limit 
																						2: value is bigger than limit 
																						3: value is equal to limit  *)               											
	Error													:	BOOL;	//Bit 6
	SyncError												:	BOOL;	//Bit 13
	TxPDOState												:	BOOL;	//Bit 14 - TRUE if NOT Valid
END_VAR
VAR
	TxPDOTgl												:	BOOL;
END_VAR

(* read analog value 																					    *)
(* resolution process image			e.g.							/ 0V = 0 / 10V = 32767 / -10V = - 32768 *)
(* or directly with NoOfDigits																	250 -> 25.0°*)
(************************************************************************************************************)

(* evaluate statusword **************************************************************************************)
	Underrange 												:= Status.0;
	Overrange												:= Status.1;
	Limit_1.0												:= Status.2;
	Limit_1.1												:= Status.3;
	Limit_2.0												:= Status.4;
	Limit_2.1												:= Status.5;
	Error													:= Status.6 OR MinValue = MaxValue AND NoOfDigits = 0;
	SyncError												:= Status.13;
	TxPDOState												:= Status.14; //TRUE if not valid
	TxPDOTgl												:= Status.15;
	
(* Scaling ******************************************************************)
	IF MaxValue <> MinValue 
	THEN
		Q 													:= Offset + Scale(In , SEL(Options.0, 0.0, -32768.0), 32767.0, MinValue , MaxValue);
		IF NoOfDigits > 0
		THEN
			Q												:= TO_FMLREAL(Q,NoOfDigits);
		END_IF
	
	ELSIF NoOfDigits > 0 (* Bsp PT100 *)
	THEN
		Q													:= Offset + TO_FMLREAL(In,NoOfDigits);
		
	ELSE  													
		Q 													:= 0.0;
	END_IF

	IF 	Error AND OutOnError <> 0.000000000000000001
	THEN
		Q													:= OutOnError;
	END_IF
(**********************************************************************************************************************)

PROPERTY PUBLIC optEnableScaleSignedValue : bool
GET
optEnableScaleSignedValue := Options.0;
END_GET
SET
Options.0 := optEnableScaleSignedValue;
END_SET
END_PROPERTY

END_FUNCTION_BLOCK

// POUs/_Miscellaneous/SEQUENCE_HDL
{attribute 'no_check'}
//Sequence handle object contains all needed variables for a state machine, like timer, state variable and error handle object
FUNCTION_BLOCK SEQUENCE_HDL
VAR_INPUT
	State													:	DINT := 0;		//Current state
	Err														:	ERROR_HDL;		//Error handle object
	Text													:	STRING := '';	//Could used for user defined texts 
END_VAR             										
VAR_OUTPUT          										
	MemSetState												:	DINT := 0;		//Memory for start state , set by method "Set"
	Busy													:	BOOL := FALSE;	//State machine is active - sets to TRUE by method "Set" and state <> 0
	Done													:	BOOL := FALSE;	//State machine sucessful finished - sets to TRUE by method "Finish" if Error handle is emnpty
	TON														:	TON := (IN := FALSE); //Use Methods to control state machine time
END_VAR             	
VAR                 	
END_VAR

;

METHOD PUBLIC abort : BOOL //Return value = TRUE - state will reset to 0 and Busy to FALSE in case state was <> 0 
VAR_INPUT
END_VAR
IF state <> 0 
THEN
	Busy 													:= FALSE;
	Done 													:= FALSE;
	     													  													
	text 													:= CONCAT('ABORTED~State:',DINT_TO_STRING(state));
	text 													:= CONCAT(text,'(SetState:');
	text 													:= CONCAT(text,DINT_TO_STRING(MemSetState));
	text 													:= CONCAT(text,')/Busy=');
	text 													:= CONCAT(text,BOOL_TO_STRING(Busy));
	text 													:= CONCAT(text,'/Done=');
	text 													:= CONCAT(text,BOOL_TO_STRING(Done));
	text 													:= CONCAT(text,'/Error=');
	text 													:= CONCAT(text,BOOL_TO_STRING(Err.flag));
	
	state													:= 0;
	Abort 													:= TRUE;
ELSE
	Abort 													:= TRUE;
END_IF
END_METHOD

METHOD PUBLIC active : BOOL //Return value = TRUE if sequence handle is active (state <> 0)
VAR_INPUT
END_VAR
Busy														:= State <> 0;
Done														:= FALSE;
Active														:= Busy;
END_METHOD

METHOD PUBLIC finish : BOOL//Return value = TRUE if state was <> 0 and Err.flag = FALSE
VAR_INPUT
END_VAR
IF state <> 0 
THEN
	Busy 													:= FALSE;
	Done 													:= NOT Err.flag;
	     													  													
	text 													:= CONCAT('FINISH~State:',DINT_TO_STRING(state));
	text 													:= CONCAT(text,'(SetState:');
	text 													:= CONCAT(text,DINT_TO_STRING(MemSetState));
	text 													:= CONCAT(text,')/Busy=');
	text 													:= CONCAT(text,BOOL_TO_STRING(Busy));
	text 													:= CONCAT(text,'/Done=');
	text 													:= CONCAT(text,BOOL_TO_STRING(Done));
	
	state													:= 0;
	Finish 													:= Done;	
ELSE
	Finish 													:= FALSE;
END_IF
END_METHOD

METHOD PUBLIC incState : BOOL //Increment State by NoOfIncrements / Result always true 
VAR_INPUT
	NoOfIncrements								:	DINT;
END_VAR
State := State + NoOfIncrements;
incState := TRUE;
END_METHOD

METHOD PUBLIC reset : BOOL //return value = TRUE if execution finished 
VAR_INPUT
END_VAR
Done 														:= FALSE;
Busy 														:= FALSE;
text 														:= CONCAT('RESET~State:',DINT_TO_STRING(state));
text 														:= CONCAT(text,'(SetState:');
text 														:= CONCAT(text,DINT_TO_STRING(MemSetState));
text 														:= CONCAT(text,')/Busy=');
text 														:= CONCAT(text,BOOL_TO_STRING(Busy));
text 														:= CONCAT(text,'/Done=');
text 														:= CONCAT(text,BOOL_TO_STRING(Done));

MemSetState := state 										:=  0;
reset 														:= TRUE;
END_METHOD

METHOD PUBLIC resetWithErrHdl : BOOL //return value = TRUE if execution finished 
VAR_INPUT
END_VAR
Reset();
Err.Reset();
ResetWithErrHdl												 := TRUE;
END_METHOD

METHOD PUBLIC set : BOOL //Set MemSetstate to state value, Return value = TRUE if sequence handle will be busy (State <> 0)
VAR_INPUT
	State													:		 DINT;
END_VAR
MemSetState 												:= THIS^.state := State;
Busy 														:= state <> 0;
Done 														:= FALSE;
Set															:= Busy;
                    										
text 														:= CONCAT('SET~State:',DINT_TO_STRING(MemSetstate));
END_METHOD

PROPERTY PUBLIC ton_BT : TIME
GET
IF ton.IN
	AND NOT ton.Q
THEN
	Ton_BT 													:= ton.PT - ton.ET;
ELSE       													
	Ton_BT 													:= T#0MS;
END_IF
END_GET
END_PROPERTY

PROPERTY PUBLIC ton_PT : TIME
GET
Ton_PT 														:= ton.PT;
END_GET
SET
PUBLIC 
VAR
END_VAR
Ton.PT 														:= Ton_PT;
END_SET
END_PROPERTY

METHOD PUBLIC tonOFF : BOOL //Return value = TRUE if execution finished
VAR_INPUT
END_VAR
TonOFF 														:= TRUE;
TON(In := FALSE);
END_METHOD

METHOD PUBLIC tonON : BOOL; //Return value = TRUE if execution finished
VAR_INPUT
END_VAR
TonON 														:= TRUE;
TON(In := TRUE);
END_METHOD

METHOD PUBLIC tonRUN : BOOL //Return value status of time (Ton.Q)
VAR_INPUT
	IN														:	BOOL;
	PT														:	TIME;
END_VAR
THIS^.TON.IN := IN;
THIS^.TON.PT := PT;
TON(IN := IN , PT := PT, Q => TonRUN);
END_METHOD

END_FUNCTION_BLOCK

// POUs/_Miscellaneous/setNoOfBits
//Returns a LWORD variable with number (no) of bits set to TRUE starting from lowest significant bit (.0)  
{attribute 'displaymode':='binary'}		
FUNCTION setNoOfBits : LWORD 
VAR_INPUT
	No														:	INT;
END_VAR
VAR
	u64														:	U_64BIT_DATATYPE;
END_VAR

IF No <= 0
THEN
	setNoOfBits												:= 0;
ELSIF No <= 32
THEN
	setNoOfBits												:= TO_LWORD((EXPT(2,No) - 1));
ELSE
	u64._DWORDs[0]											:= 16#FFFFFFFF;
	u64._DWORDs[1]											:= TO_DWORD((EXPT(2,No - 32) - 1));
	setNoOfBits												:= u64._LWORD;
END_IF

END_FUNCTION

// POUs/_Miscellaneous/TEST_FB
//Should be called after new FBs to test signal flow and behavior of PlcOpen related variables 
FUNCTION_BLOCK Test_FB
VAR_OUTPUT CONSTANT
	NO_ERR 													:	INT := 0;
 	OK														:	INT := 1;
	ERR_BUSY 												:	INT := 2;
	ERR_DONE 												:	INT := 3;	
	ERR_ERR 												:	INT := 4;
	ERR_DONE_ERROR											:	INT := 5;
	ERR_NO_SIGNAL											:	INT := 6;
END_VAR             										
VAR_INPUT           										
	Reset													:	BOOL;	//The function block will be reset with a rising edge 
	Execute													:	BOOL;	//Link with Execute of the Fb to be tested
	Busy													:	BOOL;	//link with Busy Output of FB to be tested
	Error													:	BOOL;	//link with Error Output of FB to be tested
	Done													:	BOOL;	//link with Done Output of FB to be tested
END_VAR
VAR_OUTPUT
	ErrorId			:	INT := 0;	//Error identification 
END_VAR
VAR
	state			:	INT;
END_VAR

IF Reset
THEN
	state 													:= 0;
	ErrorId 												:= NO_ERR;
ELSE

